LIN {X -0.023,Y -549.868,Z 969.397,A 0.000,B 0.000,C 90.000,E1 107.457} C_DIS
LIN {X -0.196,Y -549.764,Z 969.394,A 0.000,B 0.000,C 90.000,E1 106.913} C_DIS
LIN {X -0.171,Y -550.290,Z 969.388,A 0.000,B 0.000,C 90.000,E1 105.788} C_DIS
LIN {X 0.267,Y -551.658,Z 969.372,A 0.000,B 0.000,C 90.000,E1 102.939} C_DIS
LIN {X -0.148,Y -554.267,Z 969.355,A 0.000,B 0.000,C 90.000,E1 99.905} C_DIS
LIN {X -0.028,Y -555.925,Z 969.346,A 0.000,B 0.000,C 90.000,E1 98.219} C_DIS
LIN {X -0.088,Y -557.183,Z 969.338,A 0.000,B 0.000,C 90.000,E1 96.834} C_DIS
LIN {X -0.131,Y -558.262,Z 969.330,A 0.000,B 0.000,C 90.000,E1 95.448} C_DIS
LIN {X 0.223,Y -559.010,Z 969.324,A 0.000,B 0.000,C 90.000,E1 94.302} C_DIS
LIN {X 0.157,Y -559.871,Z 969.316,A 0.000,B 0.000,C 90.000,E1 92.922} C_DIS
LIN {X 0.071,Y -560.596,Z 969.309,A 0.000,B 0.000,C 90.000,E1 91.547} C_DIS
LIN {X -0.014,Y -561.277,Z 969.301,A 0.000,B 0.000,C 90.000,E1 90.172} C_DIS
LIN {X -0.086,Y -561.729,Z 969.293,A 0.000,B 0.000,C 90.000,E1 88.797} C_DIS
LIN {X -0.140,Y -562.027,Z 969.286,A 0.000,B 0.000,C 90.000,E1 87.421} C_DIS
LIN {X -0.191,Y -562.284,Z 969.278,A 0.000,B 0.000,C 90.000,E1 86.045} C_DIS
LIN {X -0.059,Y -562.524,Z 969.269,A 0.000,B 0.000,C 90.000,E1 84.375} C_DIS
LIN {X -0.068,Y -562.691,Z 969.261,A 0.000,B 0.000,C 90.000,E1 82.996} C_DIS
LIN {X -0.263,Y -563.143,Z 969.250,A 0.000,B 0.000,C 90.000,E1 81.084} C_DIS
LIN {X -0.020,Y -564.090,Z 969.237,A 0.000,B 0.000,C 90.000,E1 78.578} C_DIS
LIN {X 0.033,Y -565.125,Z 969.226,A 0.000,B 0.000,C 90.000,E1 76.645} C_DIS
LIN {X 0.068,Y -566.236,Z 969.217,A 0.000,B 0.000,C 90.000,E1 74.991} C_DIS
LIN {X -0.109,Y -567.560,Z 969.206,A 0.000,B 0.000,C 90.000,E1 73.087} C_DIS
LIN {X 0.129,Y -568.448,Z 969.198,A 0.000,B 0.000,C 90.000,E1 71.692} C_DIS
LIN {X 0.049,Y -569.047,Z 969.192,A 0.000,B 0.000,C 90.000,E1 70.604} C_DIS
LIN {X -0.030,Y -569.624,Z 969.186,A 0.000,B 0.000,C 90.000,E1 69.518} C_DIS
LIN {X -0.086,Y -570.280,Z 969.179,A 0.000,B 0.000,C 90.000,E1 68.156} C_DIS
LIN {X 0.054,Y -570.978,Z 969.168,A 0.000,B 0.000,C 90.000,E1 66.230} C_DIS
LIN {X 0.085,Y -571.434,Z 969.159,A 0.000,B 0.000,C 90.000,E1 64.588} C_DIS
LIN {X -0.228,Y -571.757,Z 969.151,A 0.000,B 0.000,C 90.000,E1 63.256} C_DIS
LIN {X -0.281,Y -571.994,Z 969.144,A 0.000,B 0.000,C 90.000,E1 61.897} C_DIS
LIN {X -0.054,Y -572.126,Z 969.136,A 0.000,B 0.000,C 90.000,E1 60.511} C_DIS
LIN {X -0.165,Y -572.288,Z 969.126,A 0.000,B 0.000,C 90.000,E1 58.614} C_DIS
LIN {X 0.003,Y -572.425,Z 969.117,A 0.000,B 0.000,C 90.000,E1 56.962} C_DIS
LIN {X 0.046,Y -572.265,Z 969.109,A 0.000,B 0.000,C 90.000,E1 55.595} C_DIS
LIN {X 0.130,Y -572.183,Z 969.104,A 0.000,B 0.000,C 90.000,E1 54.769} C_DIS
LIN {X -0.119,Y -571.801,Z 969.098,A 0.000,B 0.000,C 90.000,E1 53.703} C_DIS
LIN {X 0.293,Y -571.456,Z 969.094,A 0.000,B 0.000,C 90.000,E1 52.844} C_DIS
LIN {X -0.104,Y -570.939,Z 969.089,A 0.000,B 0.000,C 90.000,E1 52.065} C_DIS
LIN {X 0.104,Y -569.932,Z 969.082,A 0.000,B 0.000,C 90.000,E1 50.678} C_DIS
LIN {X 0.097,Y -568.784,Z 969.076,A 0.000,B 0.000,C 90.000,E1 49.585} C_DIS
LIN {X 0.027,Y -567.827,Z 969.071,A 0.000,B 0.000,C 90.000,E1 48.771} C_DIS
LIN {X -0.062,Y -566.696,Z 969.066,A 0.000,B 0.000,C 90.000,E1 47.957} C_DIS
LIN {X -0.203,Y -565.370,Z 969.062,A 0.000,B 0.000,C 90.000,E1 47.148} C_DIS
LIN {X -0.033,Y -564.399,Z 969.059,A 0.000,B 0.000,C 90.000,E1 46.581} C_DIS
LIN {X -0.027,Y -561.491,Z 969.051,A 0.000,B 0.000,C 90.000,E1 45.202} C_DIS
LIN {X 0.184,Y -559.483,Z 969.047,A 0.000,B 0.000,C 90.000,E1 44.352} C_DIS
LIN {X -0.025,Y -557.111,Z 969.042,A 0.000,B 0.000,C 90.000,E1 43.542} C_DIS
LIN {X 0.146,Y -554.460,Z 969.037,A 0.000,B 0.000,C 90.000,E1 42.690} C_DIS
LIN {X 0.288,Y -551.523,Z 969.033,A 0.000,B 0.000,C 90.000,E1 41.838} C_DIS
LIN {X -0.016,Y -549.373,Z 969.030,A 0.000,B 0.000,C 90.000,E1 41.310} C_DIS
LIN {X 0.027,Y -547.039,Z 969.026,A 0.000,B 0.000,C 90.000,E1 40.744} C_DIS
LIN {X -0.244,Y -541.935,Z 969.020,A 0.000,B 0.000,C 90.000,E1 39.644} C_DIS
LIN {X 0.162,Y -537.549,Z 969.015,A 0.000,B 0.000,C 90.000,E1 38.749} C_DIS
LIN {X 0.182,Y -532.876,Z 969.011,A 0.000,B 0.000,C 90.000,E1 37.890} C_DIS
LIN {X 0.154,Y -527.896,Z 969.006,A 0.000,B 0.000,C 90.000,E1 37.030} C_DIS
LIN {X 0.207,Y -521.789,Z 969.000,A 0.000,B 0.000,C 90.000,E1 36.011} C_DIS
LIN {X 0.112,Y -518.131,Z 968.997,A 0.000,B 0.000,C 90.000,E1 35.438} C_DIS
LIN {X 0.047,Y -512.314,Z 968.992,A 0.000,B 0.000,C 90.000,E1 34.565} C_DIS
LIN {X -0.019,Y -507.007,Z 968.988,A 0.000,B 0.000,C 90.000,E1 33.833} C_DIS
LIN {X -0.002,Y -501.298,Z 968.984,A 0.000,B 0.000,C 90.000,E1 33.086} C_DIS
LIN {X 0.100,Y -497.644,Z 968.981,A 0.000,B 0.000,C 90.000,E1 32.625} C_DIS
LIN {X -0.236,Y -493.784,Z 968.979,A 0.000,B 0.000,C 90.000,E1 32.212} C_DIS
LIN {X 0.054,Y -485.973,Z 968.974,A 0.000,B 0.000,C 90.000,E1 31.337} C_DIS
LIN {X -0.221,Y -480.273,Z 968.971,A 0.000,B 0.000,C 90.000,E1 30.797} C_DIS
LIN {X 0.069,Y -471.888,Z 968.966,A 0.000,B 0.000,C 90.000,E1 29.951} C_DIS
LIN {X -0.039,Y -461.755,Z 968.961,A 0.000,B 0.000,C 90.000,E1 29.027} C_DIS
LIN {X 0.120,Y -451.489,Z 968.956,A 0.000,B 0.000,C 90.000,E1 28.103} C_DIS
LIN {X 0.116,Y -436.406,Z 968.949,A 0.000,B 0.000,C 90.000,E1 26.821} C_DIS
LIN {X 0.074,Y -416.976,Z 968.939,A 0.000,B 0.000,C 90.000,E1 25.079} C_DIS
LIN {X 0.121,Y -403.934,Z 968.932,A 0.000,B 0.000,C 90.000,E1 23.770} C_DIS
LIN {X -0.172,Y -398.411,Z 968.929,A 0.000,B 0.000,C 90.000,E1 23.206} C_DIS
LIN {X 0.109,Y -395.804,Z 968.927,A 0.000,B 0.000,C 90.000,E1 22.845} C_DIS
LIN {X 0.092,Y -393.284,Z 968.925,A 0.000,B 0.000,C 90.000,E1 22.461} C_DIS
LIN {X 0.119,Y -392.305,Z 968.924,A 0.000,B 0.000,C 90.000,E1 22.280} C_DIS
LIN {X -0.046,Y -391.014,Z 968.922,A 0.000,B 0.000,C 90.000,E1 21.950} C_DIS
LIN {X -0.023,Y -390.506,Z 968.921,A 0.000,B 0.000,C 90.000,E1 21.770} C_DIS
LIN {X 0.080,Y -389.820,Z 968.918,A 0.000,B 0.000,C 90.000,E1 21.227} C_DIS
LIN {X 0.173,Y -389.839,Z 968.913,A 0.000,B 0.000,C 90.000,E1 20.301} C_DIS
LIN {X 0.011,Y -391.179,Z 968.903,A 0.000,B 0.000,C 90.000,E1 18.544} C_DIS
LIN {X -0.191,Y -393.357,Z 968.891,A 0.000,B 0.000,C 90.000,E1 16.441} C_DIS
LIN {X -0.016,Y -396.359,Z 968.878,A 0.000,B 0.000,C 90.000,E1 13.939} C_DIS
LIN {X -0.057,Y -400.300,Z 968.862,A 0.000,B 0.000,C 90.000,E1 11.130} C_DIS
LIN {X -0.098,Y -405.563,Z 968.844,A 0.000,B 0.000,C 90.000,E1 7.992} C_DIS
LIN {X -0.088,Y -410.839,Z 968.829,A 0.000,B 0.000,C 90.000,E1 5.220} C_DIS
LIN {X -0.030,Y -415.911,Z 968.816,A 0.000,B 0.000,C 90.000,E1 2.808} C_DIS
LIN {X 0.139,Y -421.480,Z 968.802,A 0.000,B 0.000,C 90.000,E1 0.401} C_DIS
LIN {X 0.000,Y -422.745,Z 968.800,A 0.000,B 0.000,C 90.000,E1 360.000} C_DIS
LIN {X 0.029,Y -424.625,Z 968.798,A 0.000,B 0.000,C 90.000,E1 359.542} C_DIS
LIN {X 0.053,Y -425.384,Z 968.797,A 0.000,B 0.000,C 90.000,E1 359.370} C_DIS
LIN {X -0.103,Y -429.458,Z 968.793,A 0.000,B 0.000,C 90.000,E1 358.797} C_DIS
LIN {X 0.126,Y -430.225,Z 968.793,A 0.000,B 0.000,C 90.000,E1 358.682} C_DIS
LIN {X 0.059,Y -434.488,Z 968.791,A 0.000,B 0.000,C 90.000,E1 358.339} C_DIS
LIN {X -0.032,Y -440.318,Z 968.789,A 0.000,B 0.000,C 90.000,E1 357.993} C_DIS
LIN {X 0.099,Y -448.688,Z 968.786,A 0.000,B 0.000,C 90.000,E1 357.535} C_DIS
LIN {X 0.144,Y -465.517,Z 968.781,A 0.000,B 0.000,C 90.000,E1 356.617} C_DIS
LIN {X -0.075,Y -475.617,Z 968.778,A 0.000,B 0.000,C 90.000,E1 356.102} C_DIS
LIN {X 0.065,Y -485.654,Z 968.775,A 0.000,B 0.000,C 90.000,E1 355.527} C_DIS
LIN {X 0.020,Y -503.780,Z 968.769,A 0.000,B 0.000,C 90.000,E1 354.489} C_DIS
LIN {X 0.137,Y -510.089,Z 968.767,A 0.000,B 0.000,C 90.000,E1 354.090} C_DIS
LIN {X -0.223,Y -519.507,Z 968.764,A 0.000,B 0.000,C 90.000,E1 353.514} C_DIS
LIN {X 0.172,Y -525.754,Z 968.762,A 0.000,B 0.000,C 90.000,E1 353.053} C_DIS
LIN {X -0.135,Y -533.195,Z 968.758,A 0.000,B 0.000,C 90.000,E1 352.527} C_DIS
LIN {X -0.243,Y -540.333,Z 968.755,A 0.000,B 0.000,C 90.000,E1 351.951} C_DIS
LIN {X -0.086,Y -547.213,Z 968.752,A 0.000,B 0.000,C 90.000,E1 351.310} C_DIS
LIN {X -0.080,Y -556.131,Z 968.747,A 0.000,B 0.000,C 90.000,E1 350.387} C_DIS
LIN {X 0.141,Y -558.635,Z 968.745,A 0.000,B 0.000,C 90.000,E1 350.095} C_DIS
LIN {X 0.222,Y -564.089,Z 968.741,A 0.000,B 0.000,C 90.000,E1 349.398} C_DIS
LIN {X -0.004,Y -568.264,Z 968.738,A 0.000,B 0.000,C 90.000,E1 348.870} C_DIS
LIN {X 0.117,Y -573.079,Z 968.734,A 0.000,B 0.000,C 90.000,E1 348.173} C_DIS
LIN {X -0.164,Y -577.486,Z 968.731,A 0.000,B 0.000,C 90.000,E1 347.521} C_DIS
LIN {X 0.031,Y -581.576,Z 968.727,A 0.000,B 0.000,C 90.000,E1 346.825} C_DIS
LIN {X 0.301,Y -586.151,Z 968.722,A 0.000,B 0.000,C 90.000,E1 345.992} C_DIS
LIN {X 0.165,Y -591.857,Z 968.716,A 0.000,B 0.000,C 90.000,E1 344.936} C_DIS
LIN {X -0.090,Y -596.515,Z 968.711,A 0.000,B 0.000,C 90.000,E1 344.031} C_DIS
LIN {X 0.122,Y -600.980,Z 968.706,A 0.000,B 0.000,C 90.000,E1 343.087} C_DIS
LIN {X -0.019,Y -605.148,Z 968.701,A 0.000,B 0.000,C 90.000,E1 342.181} C_DIS
LIN {X -0.150,Y -609.583,Z 968.695,A 0.000,B 0.000,C 90.000,E1 341.148} C_DIS
LIN {X 0.101,Y -614.858,Z 968.688,A 0.000,B 0.000,C 90.000,E1 339.826} C_DIS
LIN {X 0.316,Y -618.741,Z 968.682,A 0.000,B 0.000,C 90.000,E1 338.773} C_DIS
LIN {X -0.226,Y -623.156,Z 968.675,A 0.000,B 0.000,C 90.000,E1 337.539} C_DIS
LIN {X 0.109,Y -626.452,Z 968.669,A 0.000,B 0.000,C 90.000,E1 336.485} C_DIS
LIN {X -0.089,Y -629.658,Z 968.664,A 0.000,B 0.000,C 90.000,E1 335.485} C_DIS
LIN {X 0.055,Y -633.253,Z 968.657,A 0.000,B 0.000,C 90.000,E1 334.204} C_DIS
LIN {X -0.108,Y -635.188,Z 968.653,A 0.000,B 0.000,C 90.000,E1 333.461} C_DIS
LIN {X 0.124,Y -638.244,Z 968.646,A 0.000,B 0.000,C 90.000,E1 332.180} C_DIS
LIN {X 0.204,Y -641.584,Z 968.637,A 0.000,B 0.000,C 90.000,E1 330.667} C_DIS
LIN {X 0.222,Y -643.625,Z 968.632,A 0.000,B 0.000,C 90.000,E1 329.665} C_DIS
LIN {X 0.270,Y -645.444,Z 968.626,A 0.000,B 0.000,C 90.000,E1 328.663} C_DIS
LIN {X -0.207,Y -647.060,Z 968.621,A 0.000,B 0.000,C 90.000,E1 327.709} C_DIS
LIN {X -0.190,Y -648.192,Z 968.616,A 0.000,B 0.000,C 90.000,E1 326.962} C_DIS
LIN {X -0.096,Y -649.465,Z 968.611,A 0.000,B 0.000,C 90.000,E1 325.960} C_DIS
LIN {X 0.274,Y -650.838,Z 968.604,A 0.000,B 0.000,C 90.000,E1 324.689} C_DIS
LIN {X 0.228,Y -651.725,Z 968.599,A 0.000,B 0.000,C 90.000,E1 323.703} C_DIS
LIN {X 0.117,Y -652.636,Z 968.592,A 0.000,B 0.000,C 90.000,E1 322.477} C_DIS
LIN {X 0.020,Y -653.424,Z 968.585,A 0.000,B 0.000,C 90.000,E1 321.251} C_DIS
LIN {X 0.341,Y -654.031,Z 968.578,A 0.000,B 0.000,C 90.000,E1 319.989} C_DIS
LIN {X 0.131,Y -654.735,Z 968.570,A 0.000,B 0.000,C 90.000,E1 318.528} C_DIS
LIN {X 0.278,Y -656.513,Z 968.556,A 0.000,B 0.000,C 90.000,E1 316.053} C_DIS
LIN {X 0.182,Y -657.161,Z 968.552,A 0.000,B 0.000,C 90.000,E1 315.324} C_DIS
LIN {X -0.074,Y -658.922,Z 968.540,A 0.000,B 0.000,C 90.000,E1 313.137} C_DIS
LIN {X -0.192,Y -660.209,Z 968.531,A 0.000,B 0.000,C 90.000,E1 311.676} C_DIS
LIN {X 0.217,Y -661.294,Z 968.523,A 0.000,B 0.000,C 90.000,E1 310.172} C_DIS
LIN {X -0.254,Y -662.083,Z 968.517,A 0.000,B 0.000,C 90.000,E1 308.991} C_DIS
LIN {X 0.214,Y -662.804,Z 968.510,A 0.000,B 0.000,C 90.000,E1 307.729} C_DIS
LIN {X -0.172,Y -663.190,Z 968.506,A 0.000,B 0.000,C 90.000,E1 307.030} C_DIS
LIN {X 0.395,Y -663.564,Z 968.498,A 0.000,B 0.000,C 90.000,E1 305.518} C_DIS
LIN {X -0.171,Y -664.153,Z 968.485,A 0.000,B 0.000,C 90.000,E1 303.372} C_DIS
LIN {X -0.137,Y -666.262,Z 968.465,A 0.000,B 0.000,C 90.000,E1 299.716} C_DIS
LIN {X -0.283,Y -671.532,Z 968.444,A 0.000,B 0.000,C 90.000,E1 295.848} C_DIS
LIN {X -0.069,Y -675.006,Z 968.433,A 0.000,B 0.000,C 90.000,E1 293.898} C_DIS
LIN {X -0.239,Y -676.483,Z 968.427,A 0.000,B 0.000,C 90.000,E1 292.950} C_DIS
LIN {X -0.138,Y -676.843,Z 968.425,A 0.000,B 0.000,C 90.000,E1 292.461} C_DIS
LIN {X 0.042,Y -676.976,Z 968.423,A 0.000,B 0.000,C 90.000,E1 292.206} C_DIS
LIN {X 0.149,Y -676.527,Z 968.421,A 0.000,B 0.000,C 90.000,E1 291.716} C_DIS
LIN {X 0.078,Y -676.181,Z 968.419,A 0.000,B 0.000,C 90.000,E1 291.482} C_DIS
LIN {X 0.255,Y -675.341,Z 968.418,A 0.000,B 0.000,C 90.000,E1 291.227} C_DIS
LIN {X -0.358,Y -673.515,Z 968.416,A 0.000,B 0.000,C 90.000,E1 290.918} C_DIS
LIN {X -0.273,Y -672.787,Z 968.415,A 0.000,B 0.000,C 90.000,E1 290.791} C_DIS
LIN {X -0.192,Y -671.707,Z 968.415,A 0.000,B 0.000,C 90.000,E1 290.663} C_DIS
LIN {X -0.200,Y -665.376,Z 968.412,A 0.000,B 0.000,C 90.000,E1 290.174} C_DIS
LIN {X 0.124,Y -655.560,Z 968.409,A 0.000,B 0.000,C 90.000,E1 289.523} C_DIS
LIN {X 0.073,Y -655.528,Z 968.409,A 0.000,B 0.000,C 90.000,E1 289.523} C_DIS
LIN {X 0.233,Y -654.459,Z 968.408,A 0.000,B 0.000,C 90.000,E1 289.322} C_DIS
LIN {X 0.188,Y -654.455,Z 968.407,A 0.000,B 0.000,C 90.000,E1 289.322} C_DIS
LIN {X -0.378,Y -654.595,Z 968.407,A 0.000,B 0.000,C 90.000,E1 289.214} C_DIS
LIN {X -0.334,Y -654.907,Z 968.406,A 0.000,B 0.000,C 90.000,E1 289.087} C_DIS
LIN {X 0.205,Y -656.377,Z 968.404,A 0.000,B 0.000,C 90.000,E1 288.671} C_DIS
LIN {X 0.223,Y -659.981,Z 968.400,A 0.000,B 0.000,C 90.000,E1 288.055} C_DIS
LIN {X 0.113,Y -664.359,Z 968.396,A 0.000,B 0.000,C 90.000,E1 287.330} C_DIS
LIN {X -0.014,Y -667.594,Z 968.393,A 0.000,B 0.000,C 90.000,E1 286.732} C_DIS
LIN {X -0.249,Y -670.811,Z 968.389,A 0.000,B 0.000,C 90.000,E1 286.024} C_DIS
LIN {X 0.379,Y -673.195,Z 968.385,A 0.000,B 0.000,C 90.000,E1 285.245} C_DIS
LIN {X 0.259,Y -674.519,Z 968.382,A 0.000,B 0.000,C 90.000,E1 284.773} C_DIS
LIN {X 0.097,Y -676.009,Z 968.378,A 0.000,B 0.000,C 90.000,E1 284.064} C_DIS
LIN {X -0.051,Y -677.082,Z 968.374,A 0.000,B 0.000,C 90.000,E1 283.355} C_DIS
LIN {X -0.192,Y -677.905,Z 968.370,A 0.000,B 0.000,C 90.000,E1 282.647} C_DIS
LIN {X 0.194,Y -678.389,Z 968.366,A 0.000,B 0.000,C 90.000,E1 281.895} C_DIS
LIN {X 0.107,Y -678.463,Z 968.364,A 0.000,B 0.000,C 90.000,E1 281.422} C_DIS
LIN {X -0.030,Y -678.147,Z 968.360,A 0.000,B 0.000,C 90.000,E1 280.715} C_DIS
LIN {X -0.250,Y -677.631,Z 968.357,A 0.000,B 0.000,C 90.000,E1 280.254} C_DIS
LIN {X 0.148,Y -676.315,Z 968.353,A 0.000,B 0.000,C 90.000,E1 279.500} C_DIS
LIN {X 0.034,Y -675.184,Z 968.350,A 0.000,B 0.000,C 90.000,E1 279.029} C_DIS
LIN {X -0.196,Y -673.706,Z 968.348,A 0.000,B 0.000,C 90.000,E1 278.568} C_DIS
LIN {X 0.158,Y -670.834,Z 968.344,A 0.000,B 0.000,C 90.000,E1 277.814} C_DIS
LIN {X -0.010,Y -669.837,Z 968.342,A 0.000,B 0.000,C 90.000,E1 277.587} C_DIS
LIN {X -0.271,Y -666.765,Z 968.339,A 0.000,B 0.000,C 90.000,E1 277.004} C_DIS
LIN {X 0.017,Y -663.153,Z 968.335,A 0.000,B 0.000,C 90.000,E1 276.372} C_DIS
LIN {X -0.285,Y -659.871,Z 968.333,A 0.000,B 0.000,C 90.000,E1 275.910} C_DIS
LIN {X -0.055,Y -655.056,Z 968.329,A 0.000,B 0.000,C 90.000,E1 275.277} C_DIS
LIN {X 0.135,Y -649.688,Z 968.326,A 0.000,B 0.000,C 90.000,E1 274.645} C_DIS
LIN {X -0.192,Y -646.299,Z 968.324,A 0.000,B 0.000,C 90.000,E1 274.302} C_DIS
LIN {X 0.019,Y -640.144,Z 968.320,A 0.000,B 0.000,C 90.000,E1 273.669} C_DIS
LIN {X -0.189,Y -634.950,Z 968.318,A 0.000,B 0.000,C 90.000,E1 273.212} C_DIS
LIN {X -0.154,Y -627.970,Z 968.315,A 0.000,B 0.000,C 90.000,E1 272.636} C_DIS
LIN {X 0.018,Y -623.712,Z 968.313,A 0.000,B 0.000,C 90.000,E1 272.293} C_DIS
LIN {X -0.197,Y -617.870,Z 968.310,A 0.000,B 0.000,C 90.000,E1 271.892} C_DIS
LIN {X 0.051,Y -609.892,Z 968.308,A 0.000,B 0.000,C 90.000,E1 271.375} C_DIS
LIN {X -0.138,Y -603.402,Z 968.306,A 0.000,B 0.000,C 90.000,E1 271.031} C_DIS
LIN {X 0.234,Y -598.344,Z 968.304,A 0.000,B 0.000,C 90.000,E1 270.745} C_DIS
LIN {X 0.062,Y -591.196,Z 968.303,A 0.000,B 0.000,C 90.000,E1 270.458} C_DIS
LIN {X 0.209,Y -583.942,Z 968.301,A 0.000,B 0.000,C 90.000,E1 270.172} C_DIS
LIN {X 0.135,Y -578.187,Z 968.300,A 0.000,B 0.000,C 90.000,E1 270.000} C_DIS
LIN {X -0.099,Y -570.546,Z 968.299,A 0.000,B 0.000,C 90.000,E1 269.828} C_DIS
LIN {X -0.161,Y -564.727,Z 968.298,A 0.000,B 0.000,C 90.000,E1 269.714} C_DIS
LIN {X 0.108,Y -557.088,Z 968.298,A 0.000,B 0.000,C 90.000,E1 269.599} C_DIS
LIN {X 0.078,Y -553.455,Z 968.298,A 0.000,B 0.000,C 90.000,E1 269.599} C_DIS
LIN {X 0.049,Y -546.789,Z 968.298,A 0.000,B 0.000,C 90.000,E1 269.599} C_DIS
LIN {X -0.161,Y -543.039,Z 968.297,A 0.000,B 0.000,C 90.000,E1 269.427} C_DIS
LIN {X -0.210,Y -542.978,Z 968.297,A 0.000,B 0.000,C 90.000,E1 269.427} C_DIS
LIN {X -0.108,Y -542.551,Z 968.295,A 0.000,B 0.000,C 90.000,E1 269.026} C_DIS
LIN {X 0.062,Y -541.451,Z 968.287,A 0.000,B 0.000,C 90.000,E1 267.593} C_DIS
LIN {X 0.258,Y -540.117,Z 968.276,A 0.000,B 0.000,C 90.000,E1 265.584} C_DIS
LIN {X -0.142,Y -539.070,Z 968.268,A 0.000,B 0.000,C 90.000,E1 264.204} C_DIS
LIN {X -0.028,Y -538.231,Z 968.261,A 0.000,B 0.000,C 90.000,E1 263.053} C_DIS
LIN {X 0.199,Y -536.932,Z 968.254,A 0.000,B 0.000,C 90.000,E1 261.602} C_DIS
LIN {X -0.154,Y -535.172,Z 968.244,A 0.000,B 0.000,C 90.000,E1 259.926} C_DIS
LIN {X 0.110,Y -533.460,Z 968.236,A 0.000,B 0.000,C 90.000,E1 258.465} C_DIS
LIN {X -0.179,Y -531.773,Z 968.228,A 0.000,B 0.000,C 90.000,E1 257.061} C_DIS
LIN {X -0.154,Y -529.038,Z 968.215,A 0.000,B 0.000,C 90.000,E1 254.755} C_DIS
LIN {X 0.228,Y -527.861,Z 968.209,A 0.000,B 0.000,C 90.000,E1 253.559} C_DIS
LIN {X 0.097,Y -526.279,Z 968.201,A 0.000,B 0.000,C 90.000,E1 252.127} C_DIS
LIN {X -0.074,Y -523.664,Z 968.190,A 0.000,B 0.000,C 90.000,E1 250.115} C_DIS
LIN {X -0.101,Y -522.138,Z 968.183,A 0.000,B 0.000,C 90.000,E1 248.954} C_DIS
LIN {X -0.005,Y -520.325,Z 968.175,A 0.000,B 0.000,C 90.000,E1 247.486} C_DIS
LIN {X 0.104,Y -518.614,Z 968.168,A 0.000,B 0.000,C 90.000,E1 246.305} C_DIS
LIN {X 0.061,Y -516.427,Z 968.160,A 0.000,B 0.000,C 90.000,E1 244.845} C_DIS
LIN {X 0.098,Y -513.682,Z 968.151,A 0.000,B 0.000,C 90.000,E1 243.076} C_DIS
LIN {X -0.258,Y -511.317,Z 968.142,A 0.000,B 0.000,C 90.000,E1 241.641} C_DIS
LIN {X 0.042,Y -508.807,Z 968.134,A 0.000,B 0.000,C 90.000,E1 240.127} C_DIS
LIN {X -0.034,Y -506.572,Z 968.128,A 0.000,B 0.000,C 90.000,E1 238.948} C_DIS
LIN {X -0.003,Y -503.645,Z 968.119,A 0.000,B 0.000,C 90.000,E1 237.454} C_DIS
LIN {X -0.324,Y -501.011,Z 968.113,A 0.000,B 0.000,C 90.000,E1 236.294} C_DIS
LIN {X -0.250,Y -496.854,Z 968.103,A 0.000,B 0.000,C 90.000,E1 234.482} C_DIS
LIN {X 0.159,Y -493.558,Z 968.094,A 0.000,B 0.000,C 90.000,E1 232.924} C_DIS
LIN {X 0.254,Y -489.314,Z 968.084,A 0.000,B 0.000,C 90.000,E1 231.090} C_DIS
LIN {X 0.020,Y -484.291,Z 968.072,A 0.000,B 0.000,C 90.000,E1 228.976} C_DIS
LIN {X -0.079,Y -481.495,Z 968.065,A 0.000,B 0.000,C 90.000,E1 227.757} C_DIS
LIN {X 0.239,Y -476.090,Z 968.052,A 0.000,B 0.000,C 90.000,E1 225.243} C_DIS
LIN {X 0.089,Y -472.606,Z 968.043,A 0.000,B 0.000,C 90.000,E1 223.704} C_DIS
LIN {X 0.127,Y -469.852,Z 968.036,A 0.000,B 0.000,C 90.000,E1 222.447} C_DIS
LIN {X -0.122,Y -466.373,Z 968.027,A 0.000,B 0.000,C 90.000,E1 220.906} C_DIS
LIN {X -0.088,Y -462.897,Z 968.018,A 0.000,B 0.000,C 90.000,E1 219.322} C_DIS
LIN {X 0.068,Y -457.949,Z 968.006,A 0.000,B 0.000,C 90.000,E1 217.076} C_DIS
LIN {X 0.105,Y -454.372,Z 967.997,A 0.000,B 0.000,C 90.000,E1 215.471} C_DIS
LIN {X -0.123,Y -449.437,Z 967.985,A 0.000,B 0.000,C 90.000,E1 213.245} C_DIS
LIN {X 0.254,Y -444.521,Z 967.972,A 0.000,B 0.000,C 90.000,E1 210.924} C_DIS
LIN {X -0.120,Y -441.694,Z 967.965,A 0.000,B 0.000,C 90.000,E1 209.667} C_DIS
LIN {X -0.114,Y -438.081,Z 967.956,A 0.000,B 0.000,C 90.000,E1 208.025} C_DIS
LIN {X 0.004,Y -434.516,Z 967.946,A 0.000,B 0.000,C 90.000,E1 206.360} C_DIS
LIN {X 0.051,Y -431.526,Z 967.939,A 0.000,B 0.000,C 90.000,E1 205.027} C_DIS
LIN {X 0.046,Y -428.425,Z 967.932,A 0.000,B 0.000,C 90.000,E1 203.695} C_DIS
LIN {X -0.198,Y -423.829,Z 967.921,A 0.000,B 0.000,C 90.000,E1 201.716} C_DIS
LIN {X 0.240,Y -419.583,Z 967.909,A 0.000,B 0.000,C 90.000,E1 199.631} C_DIS
LIN {X 0.198,Y -414.058,Z 967.894,A 0.000,B 0.000,C 90.000,E1 196.913} C_DIS
LIN {X -0.112,Y -410.160,Z 967.883,A 0.000,B 0.000,C 90.000,E1 194.898} C_DIS
LIN {X -0.123,Y -406.789,Z 967.873,A 0.000,B 0.000,C 90.000,E1 193.175} C_DIS
LIN {X 0.006,Y -403.417,Z 967.864,A 0.000,B 0.000,C 90.000,E1 191.422} C_DIS
LIN {X 0.067,Y -400.132,Z 967.854,A 0.000,B 0.000,C 90.000,E1 189.670} C_DIS
LIN {X -0.071,Y -396.766,Z 967.844,A 0.000,B 0.000,C 90.000,E1 187.936} C_DIS
LIN {X -0.099,Y -391.336,Z 967.826,A 0.000,B 0.000,C 90.000,E1 184.759} C_DIS
LIN {X 0.147,Y -390.427,Z 967.822,A 0.000,B 0.000,C 90.000,E1 184.012} C_DIS
LIN {X -0.095,Y -389.546,Z 967.817,A 0.000,B 0.000,C 90.000,E1 182.980} C_DIS
LIN {X 0.115,Y -389.401,Z 967.813,A 0.000,B 0.000,C 90.000,E1 182.236} C_DIS
LIN {X 0.027,Y -389.580,Z 967.811,A 0.000,B 0.000,C 90.000,E1 181.892} C_DIS
LIN {X -0.050,Y -389.919,Z 967.809,A 0.000,B 0.000,C 90.000,E1 181.547} C_DIS
LIN {X -0.183,Y -390.765,Z 967.806,A 0.000,B 0.000,C 90.000,E1 181.031} C_DIS
LIN {X 0.082,Y -392.364,Z 967.803,A 0.000,B 0.000,C 90.000,E1 180.458} C_DIS
LIN {X 0.013,Y -394.530,Z 967.800,A 0.000,B 0.000,C 90.000,E1 179.943} C_DIS
LIN {X -0.050,Y -399.098,Z 967.796,A 0.000,B 0.000,C 90.000,E1 179.198} C_DIS
LIN {X -0.099,Y -405.521,Z 967.791,A 0.000,B 0.000,C 90.000,E1 178.453} C_DIS
LIN {X 0.081,Y -411.802,Z 967.788,A 0.000,B 0.000,C 90.000,E1 177.822} C_DIS
LIN {X -0.203,Y -419.334,Z 967.784,A 0.000,B 0.000,C 90.000,E1 177.192} C_DIS
LIN {X 0.072,Y -431.410,Z 967.778,A 0.000,B 0.000,C 90.000,E1 176.045} C_DIS
LIN {X -0.133,Y -443.385,Z 967.772,A 0.000,B 0.000,C 90.000,E1 174.951} C_DIS
LIN {X 0.180,Y -451.803,Z 967.767,A 0.000,B 0.000,C 90.000,E1 174.090} C_DIS
LIN {X -0.027,Y -458.927,Z 967.763,A 0.000,B 0.000,C 90.000,E1 173.394} C_DIS
LIN {X 0.065,Y -465.739,Z 967.759,A 0.000,B 0.000,C 90.000,E1 172.648} C_DIS
LIN {X 0.018,Y -472.498,Z 967.755,A 0.000,B 0.000,C 90.000,E1 171.894} C_DIS
LIN {X -0.232,Y -480.101,Z 967.750,A 0.000,B 0.000,C 90.000,E1 171.027} C_DIS
LIN {X 0.200,Y -489.846,Z 967.743,A 0.000,B 0.000,C 90.000,E1 169.746} C_DIS
LIN {X 0.031,Y -497.947,Z 967.737,A 0.000,B 0.000,C 90.000,E1 168.701} C_DIS
LIN {X 0.062,Y -505.525,Z 967.731,A 0.000,B 0.000,C 90.000,E1 167.645} C_DIS
LIN {X 0.023,Y -511.685,Z 967.727,A 0.000,B 0.000,C 90.000,E1 166.756} C_DIS
LIN {X -0.013,Y -513.742,Z 967.725,A 0.000,B 0.000,C 90.000,E1 166.464} C_DIS
LIN {X -0.291,Y -522.062,Z 967.717,A 0.000,B 0.000,C 90.000,E1 165.172} C_DIS
LIN {X 0.012,Y -529.357,Z 967.711,A 0.000,B 0.000,C 90.000,E1 163.976} C_DIS
LIN {X 0.121,Y -537.301,Z 967.704,A 0.000,B 0.000,C 90.000,E1 162.670} C_DIS
LIN {X -0.210,Y -548.220,Z 967.694,A 0.000,B 0.000,C 90.000,E1 160.859} C_DIS
LIN {X 0.146,Y -554.756,Z 967.687,A 0.000,B 0.000,C 90.000,E1 159.699} C_DIS
LIN {X -0.024,Y -561.770,Z 967.680,A 0.000,B 0.000,C 90.000,E1 158.465} C_DIS
LIN {X 0.105,Y -566.926,Z 967.675,A 0.000,B 0.000,C 90.000,E1 157.486} C_DIS
LIN {X 0.078,Y -571.194,Z 967.670,A 0.000,B 0.000,C 90.000,E1 156.666} C_DIS
LIN {X 0.078,Y -577.855,Z 967.663,A 0.000,B 0.000,C 90.000,E1 155.305} C_DIS
LIN {X -0.359,Y -581.485,Z 967.658,A 0.000,B 0.000,C 90.000,E1 154.537} C_DIS
LIN {X -0.105,Y -585.984,Z 967.652,A 0.000,B 0.000,C 90.000,E1 153.435} C_DIS
LIN {X -0.050,Y -590.172,Z 967.646,A 0.000,B 0.000,C 90.000,E1 152.359} C_DIS
LIN {X -0.190,Y -593.854,Z 967.641,A 0.000,B 0.000,C 90.000,E1 151.307} C_DIS
LIN {X 0.367,Y -599.028,Z 967.632,A 0.000,B 0.000,C 90.000,E1 149.665} C_DIS
LIN {X -0.167,Y -602.444,Z 967.626,A 0.000,B 0.000,C 90.000,E1 148.663} C_DIS
LIN {X 0.103,Y -606.702,Z 967.619,A 0.000,B 0.000,C 90.000,E1 147.327} C_DIS
LIN {X -0.011,Y -609.910,Z 967.613,A 0.000,B 0.000,C 90.000,E1 146.294} C_DIS
LIN {X -0.082,Y -613.296,Z 967.607,A 0.000,B 0.000,C 90.000,E1 145.261} C_DIS
LIN {X -0.003,Y -618.249,Z 967.598,A 0.000,B 0.000,C 90.000,E1 143.703} C_DIS
LIN {X 0.012,Y -623.840,Z 967.588,A 0.000,B 0.000,C 90.000,E1 141.904} C_DIS
LIN {X -0.151,Y -627.845,Z 967.581,A 0.000,B 0.000,C 90.000,E1 140.642} C_DIS
LIN {X -0.246,Y -631.776,Z 967.574,A 0.000,B 0.000,C 90.000,E1 139.380} C_DIS
LIN {X 0.304,Y -638.188,Z 967.563,A 0.000,B 0.000,C 90.000,E1 137.310} C_DIS
LIN {X 0.326,Y -642.327,Z 967.556,A 0.000,B 0.000,C 90.000,E1 136.053} C_DIS
LIN {X -0.113,Y -647.370,Z 967.548,A 0.000,B 0.000,C 90.000,E1 134.595} C_DIS
LIN {X -0.036,Y -653.433,Z 967.538,A 0.000,B 0.000,C 90.000,E1 132.852} C_DIS
LIN {X 0.172,Y -661.554,Z 967.526,A 0.000,B 0.000,C 90.000,E1 130.620} C_DIS
LIN {X 0.136,Y -666.155,Z 967.519,A 0.000,B 0.000,C 90.000,E1 129.402} C_DIS
LIN {X -0.246,Y -669.688,Z 967.514,A 0.000,B 0.000,C 90.000,E1 128.463} C_DIS
LIN {X -0.057,Y -674.761,Z 967.506,A 0.000,B 0.000,C 90.000,E1 126.996} C_DIS
LIN {X 0.213,Y -677.875,Z 967.500,A 0.000,B 0.000,C 90.000,E1 126.011} C_DIS
LIN {X 0.139,Y -681.585,Z 967.494,A 0.000,B 0.000,C 90.000,E1 124.818} C_DIS
LIN {X 0.117,Y -684.390,Z 967.488,A 0.000,B 0.000,C 90.000,E1 123.865} C_DIS
LIN {X -0.437,Y -687.004,Z 967.483,A 0.000,B 0.000,C 90.000,E1 122.959} C_DIS
LIN {X -0.387,Y -689.468,Z 967.478,A 0.000,B 0.000,C 90.000,E1 122.005} C_DIS
LIN {X 0.280,Y -691.807,Z 967.472,A 0.000,B 0.000,C 90.000,E1 121.003} C_DIS
LIN {X 0.035,Y -693.923,Z 967.467,A 0.000,B 0.000,C 90.000,E1 120.079} C_DIS
LIN {X -0.434,Y -695.321,Z 967.463,A 0.000,B 0.000,C 90.000,E1 119.411} C_DIS
LIN {X -0.029,Y -696.629,Z 967.458,A 0.000,B 0.000,C 90.000,E1 118.437} C_DIS
LIN {X 0.039,Y -697.909,Z 967.451,A 0.000,B 0.000,C 90.000,E1 117.257} C_DIS
LIN {X 0.161,Y -698.707,Z 967.446,A 0.000,B 0.000,C 90.000,E1 116.309} C_DIS
LIN {X -0.330,Y -699.277,Z 967.441,A 0.000,B 0.000,C 90.000,E1 115.412} C_DIS
LIN {X -0.161,Y -699.520,Z 967.437,A 0.000,B 0.000,C 90.000,E1 114.695} C_DIS
LIN {X 0.081,Y -699.511,Z 967.435,A 0.000,B 0.000,C 90.000,E1 114.207} C_DIS
LIN {X -0.308,Y -699.164,Z 967.432,A 0.000,B 0.000,C 90.000,E1 113.770} C_DIS
LIN {X -0.042,Y -698.683,Z 967.431,A 0.000,B 0.000,C 90.000,E1 113.515} C_DIS
LIN {X 0.207,Y -697.286,Z 967.428,A 0.000,B 0.000,C 90.000,E1 113.025} C_DIS
LIN {X -0.306,Y -696.683,Z 967.427,A 0.000,B 0.000,C 90.000,E1 112.950} C_DIS
LIN {X -0.194,Y -693.909,Z 967.425,A 0.000,B 0.000,C 90.000,E1 112.589} C_DIS
LIN {X 0.051,Y -691.862,Z 967.424,A 0.000,B 0.000,C 90.000,E1 112.333} C_DIS
LIN {X 0.170,Y -690.258,Z 967.424,A 0.000,B 0.000,C 90.000,E1 112.206} C_DIS
LIN {X 0.045,Y -685.997,Z 967.422,A 0.000,B 0.000,C 90.000,E1 112.025} C_DIS
LIN {X -0.056,Y -682.203,Z 967.422,A 0.000,B 0.000,C 90.000,E1 111.897} C_DIS
LIN {X 0.140,Y -676.018,Z 967.421,A 0.000,B 0.000,C 90.000,E1 111.716} C_DIS
LIN {X -0.109,Y -674.262,Z 967.421,A 0.000,B 0.000,C 90.000,E1 111.716} C_DIS
LIN {X 0.226,Y -667.115,Z 967.421,A 0.000,B 0.000,C 90.000,E1 111.663} C_DIS
LIN {X 0.167,Y -627.310,Z 967.420,A 0.000,B 0.000,C 90.000,E1 111.663} C_DIS
LIN {X 0.224,Y -622.838,Z 967.420,A 0.000,B 0.000,C 90.000,E1 111.589} C_DIS
LIN {X -0.100,Y -616.034,Z 967.419,A 0.000,B 0.000,C 90.000,E1 111.461} C_DIS
LIN {X -0.055,Y -609.075,Z 967.418,A 0.000,B 0.000,C 90.000,E1 111.227} C_DIS
LIN {X -0.202,Y -604.447,Z 967.417,A 0.000,B 0.000,C 90.000,E1 111.046} C_DIS
LIN {X 0.226,Y -599.289,Z 967.415,A 0.000,B 0.000,C 90.000,E1 110.737} C_DIS
LIN {X -0.097,Y -592.629,Z 967.413,A 0.000,B 0.000,C 90.000,E1 110.355} C_DIS
LIN {X 0.329,Y -583.313,Z 967.409,A 0.000,B 0.000,C 90.000,E1 109.631} C_DIS
LIN {X 0.207,Y -576.121,Z 967.406,A 0.000,B 0.000,C 90.000,E1 109.087} C_DIS
LIN {X -0.176,Y -574.529,Z 967.406,A 0.000,B 0.000,C 90.000,E1 109.014} C_DIS
LIN {X -0.017,Y -567.870,Z 967.403,A 0.000,B 0.000,C 90.000,E1 108.598} C_DIS
LIN {X 0.198,Y -552.790,Z 967.399,A 0.000,B 0.000,C 90.000,E1 107.819} C_DIS
LIN {X -0.111,Y -550.419,Z 967.398,A 0.000,B 0.000,C 90.000,E1 107.638} C_DIS
LIN {X -0.149,Y -550.391,Z 967.398,A 0.000,B 0.000,C 90.000,E1 107.638} C_DIS
LIN {X 0.177,Y -549.932,Z 967.397,A 0.000,B 0.000,C 90.000,E1 107.402} C_DIS
LIN {X -0.099,Y -549.969,Z 967.393,A 0.000,B 0.000,C 90.000,E1 106.732} C_DIS
LIN {X -0.072,Y -550.481,Z 967.387,A 0.000,B 0.000,C 90.000,E1 105.607} C_DIS
LIN {X 0.127,Y -551.713,Z 967.373,A 0.000,B 0.000,C 90.000,E1 103.063} C_DIS
LIN {X -0.051,Y -554.530,Z 967.354,A 0.000,B 0.000,C 90.000,E1 99.726} C_DIS
LIN {X 0.117,Y -556.419,Z 967.343,A 0.000,B 0.000,C 90.000,E1 97.757} C_DIS
LIN {X -0.062,Y -557.382,Z 967.337,A 0.000,B 0.000,C 90.000,E1 96.663} C_DIS
LIN {X -0.098,Y -558.452,Z 967.329,A 0.000,B 0.000,C 90.000,E1 95.277} C_DIS
LIN {X 0.263,Y -559.156,Z 967.323,A 0.000,B 0.000,C 90.000,E1 94.131} C_DIS
LIN {X 0.202,Y -560.000,Z 967.315,A 0.000,B 0.000,C 90.000,E1 92.751} C_DIS
LIN {X 0.213,Y -560.869,Z 967.306,A 0.000,B 0.000,C 90.000,E1 91.088} C_DIS
LIN {X 0.134,Y -561.465,Z 967.299,A 0.000,B 0.000,C 90.000,E1 89.714} C_DIS
LIN {X 0.063,Y -561.870,Z 967.291,A 0.000,B 0.000,C 90.000,E1 88.339} C_DIS
LIN {X 0.136,Y -562.204,Z 967.282,A 0.000,B 0.000,C 90.000,E1 86.674} C_DIS
LIN {X 0.087,Y -562.410,Z 967.274,A 0.000,B 0.000,C 90.000,E1 85.298} C_DIS
LIN {X 0.136,Y -562.633,Z 967.266,A 0.000,B 0.000,C 90.000,E1 83.913} C_DIS
LIN {X -0.051,Y -563.002,Z 967.254,A 0.000,B 0.000,C 90.000,E1 81.724} C_DIS
LIN {X -0.144,Y -563.570,Z 967.243,A 0.000,B 0.000,C 90.000,E1 79.803} C_DIS
LIN {X -0.218,Y -564.484,Z 967.233,A 0.000,B 0.000,C 90.000,E1 77.881} C_DIS
LIN {X 0.133,Y -565.807,Z 967.220,A 0.000,B 0.000,C 90.000,E1 75.644} C_DIS
LIN {X -0.053,Y -567.121,Z 967.210,A 0.000,B 0.000,C 90.000,E1 73.740} C_DIS
LIN {X 0.005,Y -568.048,Z 967.202,A 0.000,B 0.000,C 90.000,E1 72.362} C_DIS
LIN {X -0.126,Y -569.029,Z 967.193,A 0.000,B 0.000,C 90.000,E1 70.732} C_DIS
LIN {X 0.138,Y -569.701,Z 967.185,A 0.000,B 0.000,C 90.000,E1 69.337} C_DIS
LIN {X 0.082,Y -570.331,Z 967.178,A 0.000,B 0.000,C 90.000,E1 67.975} C_DIS
LIN {X 0.218,Y -571.002,Z 967.167,A 0.000,B 0.000,C 90.000,E1 66.049} C_DIS
LIN {X 0.245,Y -571.396,Z 967.158,A 0.000,B 0.000,C 90.000,E1 64.409} C_DIS
LIN {X -0.075,Y -571.717,Z 967.150,A 0.000,B 0.000,C 90.000,E1 63.076} C_DIS
LIN {X -0.136,Y -571.932,Z 967.143,A 0.000,B 0.000,C 90.000,E1 61.719} C_DIS
LIN {X 0.083,Y -572.044,Z 967.135,A 0.000,B 0.000,C 90.000,E1 60.333} C_DIS
LIN {X -0.184,Y -572.179,Z 967.128,A 0.000,B 0.000,C 90.000,E1 58.997} C_DIS
LIN {X 0.339,Y -572.294,Z 967.120,A 0.000,B 0.000,C 90.000,E1 57.582} C_DIS
LIN {X 0.113,Y -572.300,Z 967.116,A 0.000,B 0.000,C 90.000,E1 56.786} C_DIS
LIN {X -0.004,Y -572.115,Z 967.108,A 0.000,B 0.000,C 90.000,E1 55.435} C_DIS
LIN {X 0.082,Y -571.976,Z 967.103,A 0.000,B 0.000,C 90.000,E1 54.609} C_DIS
LIN {X 0.022,Y -571.868,Z 967.100,A 0.000,B 0.000,C 90.000,E1 54.069} C_DIS
LIN {X 0.111,Y -571.359,Z 967.094,A 0.000,B 0.000,C 90.000,E1 52.970} C_DIS
LIN {X -0.283,Y -570.858,Z 967.090,A 0.000,B 0.000,C 90.000,E1 52.190} C_DIS
LIN {X -0.069,Y -569.815,Z 967.082,A 0.000,B 0.000,C 90.000,E1 50.803} C_DIS
LIN {X -0.008,Y -568.693,Z 967.076,A 0.000,B 0.000,C 90.000,E1 49.703} C_DIS
LIN {X -0.023,Y -567.363,Z 967.070,A 0.000,B 0.000,C 90.000,E1 48.609} C_DIS
LIN {X -0.049,Y -565.736,Z 967.064,A 0.000,B 0.000,C 90.000,E1 47.514} C_DIS
LIN {X 0.314,Y -563.722,Z 967.058,A 0.000,B 0.000,C 90.000,E1 46.377} C_DIS
LIN {X -0.324,Y -562.595,Z 967.055,A 0.000,B 0.000,C 90.000,E1 45.891} C_DIS
LIN {X 0.296,Y -560.732,Z 967.050,A 0.000,B 0.000,C 90.000,E1 45.000} C_DIS
LIN {X 0.102,Y -558.590,Z 967.046,A 0.000,B 0.000,C 90.000,E1 44.190} C_DIS
LIN {X -0.115,Y -556.135,Z 967.041,A 0.000,B 0.000,C 90.000,E1 43.380} C_DIS
LIN {X 0.044,Y -553.399,Z 967.036,A 0.000,B 0.000,C 90.000,E1 42.528} C_DIS
LIN {X -0.248,Y -551.394,Z 967.033,A 0.000,B 0.000,C 90.000,E1 42.000} C_DIS
LIN {X -0.136,Y -548.146,Z 967.029,A 0.000,B 0.000,C 90.000,E1 41.148} C_DIS
LIN {X -0.264,Y -545.063,Z 967.025,A 0.000,B 0.000,C 90.000,E1 40.458} C_DIS
LIN {X -0.006,Y -541.829,Z 967.021,A 0.000,B 0.000,C 90.000,E1 39.725} C_DIS
LIN {X -0.184,Y -536.672,Z 967.015,A 0.000,B 0.000,C 90.000,E1 38.749} C_DIS
LIN {X -0.171,Y -531.920,Z 967.010,A 0.000,B 0.000,C 90.000,E1 37.890} C_DIS
LIN {X 0.113,Y -526.875,Z 967.006,A 0.000,B 0.000,C 90.000,E1 36.996} C_DIS
LIN {X -0.159,Y -520.696,Z 967.000,A 0.000,B 0.000,C 90.000,E1 36.011} C_DIS
LIN {X 0.101,Y -515.084,Z 966.995,A 0.000,B 0.000,C 90.000,E1 35.105} C_DIS
LIN {X -0.228,Y -510.035,Z 966.991,A 0.000,B 0.000,C 90.000,E1 34.405} C_DIS
LIN {X 0.103,Y -504.514,Z 966.987,A 0.000,B 0.000,C 90.000,E1 33.627} C_DIS
LIN {X 0.023,Y -499.837,Z 966.984,A 0.000,B 0.000,C 90.000,E1 33.038} C_DIS
LIN {X -0.021,Y -493.605,Z 966.979,A 0.000,B 0.000,C 90.000,E1 32.291} C_DIS
LIN {X 0.238,Y -484.140,Z 966.974,A 0.000,B 0.000,C 90.000,E1 31.258} C_DIS
LIN {X -0.096,Y -476.951,Z 966.970,A 0.000,B 0.000,C 90.000,E1 30.590} C_DIS
LIN {X 0.062,Y -468.229,Z 966.965,A 0.000,B 0.000,C 90.000,E1 29.745} C_DIS
LIN {X 0.037,Y -462.348,Z 966.962,A 0.000,B 0.000,C 90.000,E1 29.205} C_DIS
LIN {X 0.024,Y -453.290,Z 966.958,A 0.000,B 0.000,C 90.000,E1 28.409} C_DIS
LIN {X -0.123,Y -441.071,Z 966.952,A 0.000,B 0.000,C 90.000,E1 27.385} C_DIS
LIN {X 0.169,Y -416.994,Z 966.940,A 0.000,B 0.000,C 90.000,E1 25.207} C_DIS
LIN {X -0.033,Y -402.378,Z 966.932,A 0.000,B 0.000,C 90.000,E1 23.770} C_DIS
LIN {X -0.192,Y -398.273,Z 966.930,A 0.000,B 0.000,C 90.000,E1 23.334} C_DIS
LIN {X 0.081,Y -396.073,Z 966.928,A 0.000,B 0.000,C 90.000,E1 23.025} C_DIS
LIN {X -0.203,Y -392.270,Z 966.925,A 0.000,B 0.000,C 90.000,E1 22.461} C_DIS
LIN {X -0.107,Y -390.513,Z 966.922,A 0.000,B 0.000,C 90.000,E1 21.950} C_DIS
LIN {X 0.220,Y -389.751,Z 966.918,A 0.000,B 0.000,C 90.000,E1 21.280} C_DIS
LIN {X 0.150,Y -389.747,Z 966.914,A 0.000,B 0.000,C 90.000,E1 20.556} C_DIS
LIN {X 0.035,Y -390.410,Z 966.908,A 0.000,B 0.000,C 90.000,E1 19.504} C_DIS
LIN {X -0.096,Y -393.983,Z 966.889,A 0.000,B 0.000,C 90.000,E1 15.969} C_DIS
LIN {X 0.040,Y -396.607,Z 966.877,A 0.000,B 0.000,C 90.000,E1 13.828} C_DIS
LIN {X 0.078,Y -401.105,Z 966.859,A 0.000,B 0.000,C 90.000,E1 10.658} C_DIS
LIN {X 0.050,Y -405.842,Z 966.844,A 0.000,B 0.000,C 90.000,E1 7.871} C_DIS
LIN {X -0.002,Y -410.468,Z 966.830,A 0.000,B 0.000,C 90.000,E1 5.454} C_DIS
LIN {X 0.090,Y -416.215,Z 966.815,A 0.000,B 0.000,C 90.000,E1 2.694} C_DIS
LIN {X -0.186,Y -420.853,Z 966.804,A 0.000,B 0.000,C 90.000,E1 0.688} C_DIS
LIN {X 0.000,Y -422.713,Z 966.800,A 0.000,B 0.000,C 90.000,E1 360.000} C_DIS
LIN {X 0.033,Y -425.462,Z 966.796,A 0.000,B 0.000,C 90.000,E1 359.312} C_DIS
LIN {X 0.085,Y -427.570,Z 966.794,A 0.000,B 0.000,C 90.000,E1 358.969} C_DIS
LIN {X -0.085,Y -429.363,Z 966.793,A 0.000,B 0.000,C 90.000,E1 358.740} C_DIS
LIN {X 0.145,Y -430.132,Z 966.793,A 0.000,B 0.000,C 90.000,E1 358.625} C_DIS
LIN {X -0.042,Y -435.272,Z 966.790,A 0.000,B 0.000,C 90.000,E1 358.224} C_DIS
LIN {X -0.087,Y -441.202,Z 966.788,A 0.000,B 0.000,C 90.000,E1 357.879} C_DIS
LIN {X 0.035,Y -447.491,Z 966.786,A 0.000,B 0.000,C 90.000,E1 357.535} C_DIS
LIN {X 0.042,Y -464.462,Z 966.781,A 0.000,B 0.000,C 90.000,E1 356.617} C_DIS
LIN {X -0.169,Y -474.565,Z 966.778,A 0.000,B 0.000,C 90.000,E1 356.102} C_DIS
LIN {X -0.046,Y -487.628,Z 966.774,A 0.000,B 0.000,C 90.000,E1 355.355} C_DIS
LIN {X -0.166,Y -502.053,Z 966.770,A 0.000,B 0.000,C 90.000,E1 354.546} C_DIS
LIN {X -0.136,Y -506.871,Z 966.768,A 0.000,B 0.000,C 90.000,E1 354.261} C_DIS
LIN {X -0.237,Y -517.773,Z 966.764,A 0.000,B 0.000,C 90.000,E1 353.571} C_DIS
LIN {X -0.274,Y -525.578,Z 966.761,A 0.000,B 0.000,C 90.000,E1 353.053} C_DIS
LIN {X 0.003,Y -533.005,Z 966.758,A 0.000,B 0.000,C 90.000,E1 352.470} C_DIS
LIN {X -0.239,Y -541.561,Z 966.754,A 0.000,B 0.000,C 90.000,E1 351.781} C_DIS
LIN {X 0.030,Y -547.048,Z 966.751,A 0.000,B 0.000,C 90.000,E1 351.254} C_DIS
LIN {X 0.179,Y -554.852,Z 966.747,A 0.000,B 0.000,C 90.000,E1 350.443} C_DIS
LIN {X 0.165,Y -558.614,Z 966.745,A 0.000,B 0.000,C 90.000,E1 350.038} C_DIS
LIN {X 0.205,Y -564.176,Z 966.741,A 0.000,B 0.000,C 90.000,E1 349.342} C_DIS
LIN {X -0.021,Y -568.361,Z 966.738,A 0.000,B 0.000,C 90.000,E1 348.814} C_DIS
LIN {X -0.218,Y -572.256,Z 966.735,A 0.000,B 0.000,C 90.000,E1 348.285} C_DIS
LIN {X -0.183,Y -577.626,Z 966.730,A 0.000,B 0.000,C 90.000,E1 347.465} C_DIS
LIN {X -0.194,Y -583.300,Z 966.725,A 0.000,B 0.000,C 90.000,E1 346.520} C_DIS
LIN {X 0.059,Y -587.023,Z 966.721,A 0.000,B 0.000,C 90.000,E1 345.825} C_DIS
LIN {X 0.311,Y -592.041,Z 966.716,A 0.000,B 0.000,C 90.000,E1 344.866} C_DIS
LIN {X -0.097,Y -596.740,Z 966.711,A 0.000,B 0.000,C 90.000,E1 343.976} C_DIS
LIN {X 0.059,Y -601.798,Z 966.705,A 0.000,B 0.000,C 90.000,E1 342.906} C_DIS
LIN {X -0.073,Y -605.918,Z 966.700,A 0.000,B 0.000,C 90.000,E1 342.000} C_DIS
LIN {X -0.193,Y -610.349,Z 966.694,A 0.000,B 0.000,C 90.000,E1 340.967} C_DIS
LIN {X -0.251,Y -614.571,Z 966.688,A 0.000,B 0.000,C 90.000,E1 339.934} C_DIS
LIN {X -0.257,Y -618.520,Z 966.683,A 0.000,B 0.000,C 90.000,E1 338.901} C_DIS
LIN {X 0.013,Y -622.148,Z 966.677,A 0.000,B 0.000,C 90.000,E1 337.847} C_DIS
LIN {X 0.337,Y -625.517,Z 966.671,A 0.000,B 0.000,C 90.000,E1 336.794} C_DIS
LIN {X 0.150,Y -629.567,Z 966.664,A 0.000,B 0.000,C 90.000,E1 335.537} C_DIS
LIN {X -0.040,Y -631.776,Z 966.660,A 0.000,B 0.000,C 90.000,E1 334.793} C_DIS
LIN {X 0.100,Y -634.597,Z 966.654,A 0.000,B 0.000,C 90.000,E1 333.768} C_DIS
LIN {X -0.236,Y -637.683,Z 966.647,A 0.000,B 0.000,C 90.000,E1 332.538} C_DIS
LIN {X -0.017,Y -639.976,Z 966.642,A 0.000,B 0.000,C 90.000,E1 331.513} C_DIS
LIN {X 0.042,Y -642.758,Z 966.635,A 0.000,B 0.000,C 90.000,E1 330.255} C_DIS
LIN {X 0.081,Y -644.706,Z 966.629,A 0.000,B 0.000,C 90.000,E1 329.253} C_DIS
LIN {X 0.217,Y -646.860,Z 966.622,A 0.000,B 0.000,C 90.000,E1 327.995} C_DIS
LIN {X -0.243,Y -648.420,Z 966.617,A 0.000,B 0.000,C 90.000,E1 327.041} C_DIS
LIN {X 0.215,Y -649.704,Z 966.611,A 0.000,B 0.000,C 90.000,E1 326.008} C_DIS
LIN {X -0.245,Y -651.385,Z 966.603,A 0.000,B 0.000,C 90.000,E1 324.562} C_DIS
LIN {X 0.098,Y -652.249,Z 966.598,A 0.000,B 0.000,C 90.000,E1 323.543} C_DIS
LIN {X 0.069,Y -652.968,Z 966.592,A 0.000,B 0.000,C 90.000,E1 322.557} C_DIS
LIN {X -0.026,Y -653.804,Z 966.585,A 0.000,B 0.000,C 90.000,E1 321.331} C_DIS
LIN {X 0.299,Y -654.457,Z 966.578,A 0.000,B 0.000,C 90.000,E1 320.070} C_DIS
LIN {X 0.065,Y -655.391,Z 966.567,A 0.000,B 0.000,C 90.000,E1 318.119} C_DIS
LIN {X 0.252,Y -656.869,Z 966.556,A 0.000,B 0.000,C 90.000,E1 316.134} C_DIS
LIN {X 0.131,Y -657.706,Z 966.551,A 0.000,B 0.000,C 90.000,E1 315.162} C_DIS
LIN {X -0.085,Y -659.307,Z 966.540,A 0.000,B 0.000,C 90.000,E1 313.218} C_DIS
LIN {X -0.194,Y -660.623,Z 966.532,A 0.000,B 0.000,C 90.000,E1 311.757} C_DIS
LIN {X 0.200,Y -661.896,Z 966.522,A 0.000,B 0.000,C 90.000,E1 310.011} C_DIS
LIN {X -0.266,Y -662.685,Z 966.516,A 0.000,B 0.000,C 90.000,E1 308.830} C_DIS
LIN {X -0.198,Y -663.393,Z 966.509,A 0.000,B 0.000,C 90.000,E1 307.604} C_DIS
LIN {X 0.261,Y -663.681,Z 966.506,A 0.000,B 0.000,C 90.000,E1 307.076} C_DIS
LIN {X -0.053,Y -664.030,Z 966.499,A 0.000,B 0.000,C 90.000,E1 305.884} C_DIS
LIN {X 0.023,Y -664.268,Z 966.493,A 0.000,B 0.000,C 90.000,E1 304.659} C_DIS
LIN {X -0.167,Y -664.746,Z 966.484,A 0.000,B 0.000,C 90.000,E1 303.214} C_DIS
LIN {X -0.028,Y -666.727,Z 966.466,A 0.000,B 0.000,C 90.000,E1 299.795} C_DIS
LIN {X 0.093,Y -670.359,Z 966.449,A 0.000,B 0.000,C 90.000,E1 296.873} C_DIS
LIN {X 0.198,Y -674.975,Z 966.435,A 0.000,B 0.000,C 90.000,E1 294.207} C_DIS
LIN {X 0.027,Y -676.537,Z 966.429,A 0.000,B 0.000,C 90.000,E1 293.259} C_DIS
LIN {X 0.127,Y -677.201,Z 966.427,A 0.000,B 0.000,C 90.000,E1 292.770} C_DIS
LIN {X 0.235,Y -677.460,Z 966.424,A 0.000,B 0.000,C 90.000,E1 292.280} C_DIS
LIN {X -0.211,Y -677.405,Z 966.423,A 0.000,B 0.000,C 90.000,E1 292.078} C_DIS
LIN {X -0.101,Y -676.870,Z 966.420,A 0.000,B 0.000,C 90.000,E1 291.589} C_DIS
LIN {X -0.170,Y -676.148,Z 966.419,A 0.000,B 0.000,C 90.000,E1 291.354} C_DIS
LIN {X -0.063,Y -673.639,Z 966.416,A 0.000,B 0.000,C 90.000,E1 290.865} C_DIS
LIN {X 0.020,Y -672.860,Z 966.415,A 0.000,B 0.000,C 90.000,E1 290.737} C_DIS
LIN {X 0.102,Y -671.703,Z 966.415,A 0.000,B 0.000,C 90.000,E1 290.610} C_DIS
LIN {X 0.025,Y -665.742,Z 966.412,A 0.000,B 0.000,C 90.000,E1 290.174} C_DIS
LIN {X -0.034,Y -657.922,Z 966.409,A 0.000,B 0.000,C 90.000,E1 289.685} C_DIS
LIN {X 0.052,Y -655.810,Z 966.409,A 0.000,B 0.000,C 90.000,E1 289.523} C_DIS
LIN {X 0.236,Y -655.776,Z 966.409,A 0.000,B 0.000,C 90.000,E1 289.504} C_DIS
LIN {X 0.114,Y -655.114,Z 966.408,A 0.000,B 0.000,C 90.000,E1 289.396} C_DIS
LIN {X 0.077,Y -655.111,Z 966.408,A 0.000,B 0.000,C 90.000,E1 289.396} C_DIS
LIN {X -0.052,Y -655.374,Z 966.406,A 0.000,B 0.000,C 90.000,E1 289.141} C_DIS
LIN {X -0.089,Y -657.393,Z 966.404,A 0.000,B 0.000,C 90.000,E1 288.652} C_DIS
LIN {X 0.151,Y -663.972,Z 966.398,A 0.000,B 0.000,C 90.000,E1 287.528} C_DIS
LIN {X 0.223,Y -667.288,Z 966.394,A 0.000,B 0.000,C 90.000,E1 286.913} C_DIS
LIN {X 0.141,Y -668.556,Z 966.393,A 0.000,B 0.000,C 90.000,E1 286.677} C_DIS
LIN {X -0.081,Y -671.681,Z 966.389,A 0.000,B 0.000,C 90.000,E1 285.969} C_DIS
LIN {X -0.031,Y -673.292,Z 966.386,A 0.000,B 0.000,C 90.000,E1 285.481} C_DIS
LIN {X -0.207,Y -675.307,Z 966.382,A 0.000,B 0.000,C 90.000,E1 284.773} C_DIS
LIN {X 0.293,Y -676.756,Z 966.378,A 0.000,B 0.000,C 90.000,E1 284.008} C_DIS
LIN {X 0.110,Y -678.173,Z 966.373,A 0.000,B 0.000,C 90.000,E1 283.063} C_DIS
LIN {X -0.021,Y -678.860,Z 966.369,A 0.000,B 0.000,C 90.000,E1 282.355} C_DIS
LIN {X -0.107,Y -679.150,Z 966.366,A 0.000,B 0.000,C 90.000,E1 281.883} C_DIS
LIN {X -0.328,Y -679.222,Z 966.363,A 0.000,B 0.000,C 90.000,E1 281.422} C_DIS
LIN {X 0.209,Y -678.872,Z 966.359,A 0.000,B 0.000,C 90.000,E1 280.658} C_DIS
LIN {X -0.006,Y -678.370,Z 966.357,A 0.000,B 0.000,C 90.000,E1 280.197} C_DIS
LIN {X -0.102,Y -677.546,Z 966.354,A 0.000,B 0.000,C 90.000,E1 279.726} C_DIS
LIN {X -0.320,Y -676.513,Z 966.351,A 0.000,B 0.000,C 90.000,E1 279.265} C_DIS
LIN {X 0.128,Y -675.136,Z 966.349,A 0.000,B 0.000,C 90.000,E1 278.746} C_DIS
LIN {X 0.066,Y -674.344,Z 966.347,A 0.000,B 0.000,C 90.000,E1 278.511} C_DIS
LIN {X -0.237,Y -671.489,Z 966.343,A 0.000,B 0.000,C 90.000,E1 277.814} C_DIS
LIN {X 0.261,Y -670.475,Z 966.342,A 0.000,B 0.000,C 90.000,E1 277.530} C_DIS
LIN {X -0.084,Y -666.675,Z 966.338,A 0.000,B 0.000,C 90.000,E1 276.834} C_DIS
LIN {X 0.297,Y -663.760,Z 966.335,A 0.000,B 0.000,C 90.000,E1 276.315} C_DIS
LIN {X -0.002,Y -660.469,Z 966.333,A 0.000,B 0.000,C 90.000,E1 275.853} C_DIS
LIN {X 0.232,Y -655.698,Z 966.329,A 0.000,B 0.000,C 90.000,E1 275.220} C_DIS
LIN {X -0.119,Y -651.460,Z 966.326,A 0.000,B 0.000,C 90.000,E1 274.759} C_DIS
LIN {X -0.008,Y -645.703,Z 966.323,A 0.000,B 0.000,C 90.000,E1 274.131} C_DIS
LIN {X -0.189,Y -640.949,Z 966.320,A 0.000,B 0.000,C 90.000,E1 273.669} C_DIS
LIN {X 0.203,Y -635.736,Z 966.318,A 0.000,B 0.000,C 90.000,E1 273.154} C_DIS
LIN {X 0.277,Y -630.311,Z 966.315,A 0.000,B 0.000,C 90.000,E1 272.694} C_DIS
LIN {X -0.153,Y -624.701,Z 966.313,A 0.000,B 0.000,C 90.000,E1 272.293} C_DIS
LIN {X 0.189,Y -618.740,Z 966.310,A 0.000,B 0.000,C 90.000,E1 271.835} C_DIS
LIN {X -0.172,Y -610.955,Z 966.308,A 0.000,B 0.000,C 90.000,E1 271.375} C_DIS
LIN {X 0.211,Y -604.474,Z 966.306,A 0.000,B 0.000,C 90.000,E1 270.974} C_DIS
LIN {X -0.282,Y -597.700,Z 966.304,A 0.000,B 0.000,C 90.000,E1 270.688} C_DIS
LIN {X 0.263,Y -590.751,Z 966.302,A 0.000,B 0.000,C 90.000,E1 270.344} C_DIS
LIN {X -0.015,Y -585.513,Z 966.301,A 0.000,B 0.000,C 90.000,E1 270.172} C_DIS
LIN {X -0.120,Y -578.006,Z 966.300,A 0.000,B 0.000,C 90.000,E1 269.943} C_DIS
LIN {X 0.035,Y -572.045,Z 966.299,A 0.000,B 0.000,C 90.000,E1 269.771} C_DIS
LIN {X -0.102,Y -565.986,Z 966.298,A 0.000,B 0.000,C 90.000,E1 269.656} C_DIS
LIN {X -0.245,Y -560.893,Z 966.298,A 0.000,B 0.000,C 90.000,E1 269.599} C_DIS
LIN {X -0.089,Y -557.236,Z 966.297,A 0.000,B 0.000,C 90.000,E1 269.542} C_DIS
LIN {X -0.146,Y -552.113,Z 966.297,A 0.000,B 0.000,C 90.000,E1 269.542} C_DIS
LIN {X -0.193,Y -547.053,Z 966.297,A 0.000,B 0.000,C 90.000,E1 269.542} C_DIS
LIN {X 0.127,Y -543.096,Z 966.296,A 0.000,B 0.000,C 90.000,E1 269.312} C_DIS
LIN {X 0.079,Y -543.016,Z 966.296,A 0.000,B 0.000,C 90.000,E1 269.312} C_DIS
LIN {X 0.061,Y -542.666,Z 966.295,A 0.000,B 0.000,C 90.000,E1 269.026} C_DIS
LIN {X -0.140,Y -542.146,Z 966.291,A 0.000,B 0.000,C 90.000,E1 268.339} C_DIS
LIN {X 0.135,Y -540.298,Z 966.277,A 0.000,B 0.000,C 90.000,E1 265.755} C_DIS
LIN {X -0.258,Y -539.291,Z 966.269,A 0.000,B 0.000,C 90.000,E1 264.375} C_DIS
LIN {X -0.136,Y -538.473,Z 966.262,A 0.000,B 0.000,C 90.000,E1 263.223} C_DIS
LIN {X 0.022,Y -537.225,Z 966.254,A 0.000,B 0.000,C 90.000,E1 261.781} C_DIS
LIN {X 0.231,Y -535.738,Z 966.246,A 0.000,B 0.000,C 90.000,E1 260.330} C_DIS
LIN {X -0.070,Y -534.468,Z 966.240,A 0.000,B 0.000,C 90.000,E1 259.218} C_DIS
LIN {X -0.237,Y -532.077,Z 966.229,A 0.000,B 0.000,C 90.000,E1 257.229} C_DIS
LIN {X -0.188,Y -529.307,Z 966.216,A 0.000,B 0.000,C 90.000,E1 254.921} C_DIS
LIN {X 0.076,Y -527.794,Z 966.208,A 0.000,B 0.000,C 90.000,E1 253.449} C_DIS
LIN {X 0.099,Y -526.173,Z 966.200,A 0.000,B 0.000,C 90.000,E1 252.000} C_DIS
LIN {X 0.260,Y -523.940,Z 966.190,A 0.000,B 0.000,C 90.000,E1 250.242} C_DIS
LIN {X 0.234,Y -522.442,Z 966.184,A 0.000,B 0.000,C 90.000,E1 249.082} C_DIS
LIN {X 0.002,Y -520.217,Z 966.174,A 0.000,B 0.000,C 90.000,E1 247.358} C_DIS
LIN {X -0.084,Y -517.628,Z 966.164,A 0.000,B 0.000,C 90.000,E1 245.613} C_DIS
LIN {X 0.195,Y -515.807,Z 966.158,A 0.000,B 0.000,C 90.000,E1 244.409} C_DIS
LIN {X -0.010,Y -513.084,Z 966.148,A 0.000,B 0.000,C 90.000,E1 242.666} C_DIS
LIN {X 0.082,Y -510.668,Z 966.140,A 0.000,B 0.000,C 90.000,E1 241.179} C_DIS
LIN {X 0.038,Y -508.651,Z 966.133,A 0.000,B 0.000,C 90.000,E1 239.999} C_DIS
LIN {X -0.043,Y -506.408,Z 966.127,A 0.000,B 0.000,C 90.000,E1 238.820} C_DIS
LIN {X -0.328,Y -504.034,Z 966.120,A 0.000,B 0.000,C 90.000,E1 237.661} C_DIS
LIN {X 0.054,Y -501.452,Z 966.114,A 0.000,B 0.000,C 90.000,E1 236.421} C_DIS
LIN {X 0.139,Y -497.302,Z 966.104,A 0.000,B 0.000,C 90.000,E1 234.609} C_DIS
LIN {X -0.274,Y -493.293,Z 966.093,A 0.000,B 0.000,C 90.000,E1 232.844} C_DIS
LIN {X -0.179,Y -489.078,Z 966.083,A 0.000,B 0.000,C 90.000,E1 231.009} C_DIS
LIN {X -0.046,Y -484.094,Z 966.071,A 0.000,B 0.000,C 90.000,E1 228.852} C_DIS
LIN {X 0.101,Y -479.870,Z 966.061,A 0.000,B 0.000,C 90.000,E1 226.986} C_DIS
LIN {X -0.194,Y -475.838,Z 966.051,A 0.000,B 0.000,C 90.000,E1 225.162} C_DIS
LIN {X -0.004,Y -472.364,Z 966.042,A 0.000,B 0.000,C 90.000,E1 223.581} C_DIS
LIN {X 0.271,Y -470.314,Z 966.037,A 0.000,B 0.000,C 90.000,E1 222.609} C_DIS
LIN {X 0.032,Y -466.827,Z 966.028,A 0.000,B 0.000,C 90.000,E1 221.067} C_DIS
LIN {X 0.075,Y -463.399,Z 966.019,A 0.000,B 0.000,C 90.000,E1 219.483} C_DIS
LIN {X -0.013,Y -457.731,Z 966.005,A 0.000,B 0.000,C 90.000,E1 216.950} C_DIS
LIN {X 0.012,Y -453.410,Z 965.995,A 0.000,B 0.000,C 90.000,E1 215.025} C_DIS
LIN {X 0.043,Y -449.179,Z 965.984,A 0.000,B 0.000,C 90.000,E1 213.086} C_DIS
LIN {X 0.172,Y -444.328,Z 965.971,A 0.000,B 0.000,C 90.000,E1 210.797} C_DIS
LIN {X -0.066,Y -439.318,Z 965.959,A 0.000,B 0.000,C 90.000,E1 208.537} C_DIS
LIN {X 0.091,Y -435.010,Z 965.948,A 0.000,B 0.000,C 90.000,E1 206.539} C_DIS
LIN {X 0.141,Y -432.060,Z 965.940,A 0.000,B 0.000,C 90.000,E1 205.207} C_DIS
LIN {X -0.032,Y -428.963,Z 965.933,A 0.000,B 0.000,C 90.000,E1 203.898} C_DIS
LIN {X 0.067,Y -422.187,Z 965.916,A 0.000,B 0.000,C 90.000,E1 200.865} C_DIS
LIN {X -0.236,Y -418.639,Z 965.907,A 0.000,B 0.000,C 90.000,E1 199.214} C_DIS
LIN {X -0.046,Y -413.843,Z 965.893,A 0.000,B 0.000,C 90.000,E1 196.804} C_DIS
LIN {X 0.131,Y -410.577,Z 965.884,A 0.000,B 0.000,C 90.000,E1 195.064} C_DIS
LIN {X 0.024,Y -407.195,Z 965.874,A 0.000,B 0.000,C 90.000,E1 193.355} C_DIS
LIN {X 0.156,Y -404.499,Z 965.867,A 0.000,B 0.000,C 90.000,E1 191.951} C_DIS
LIN {X -0.158,Y -400.532,Z 965.855,A 0.000,B 0.000,C 90.000,E1 189.905} C_DIS
LIN {X 0.144,Y -396.479,Z 965.843,A 0.000,B 0.000,C 90.000,E1 187.757} C_DIS
LIN {X -0.030,Y -390.575,Z 965.824,A 0.000,B 0.000,C 90.000,E1 184.245} C_DIS
LIN {X 0.123,Y -389.352,Z 965.818,A 0.000,B 0.000,C 90.000,E1 183.154} C_DIS
LIN {X -0.036,Y -388.970,Z 965.814,A 0.000,B 0.000,C 90.000,E1 182.465} C_DIS
LIN {X 0.139,Y -389.172,Z 965.809,A 0.000,B 0.000,C 90.000,E1 181.547} C_DIS
LIN {X 0.004,Y -389.820,Z 965.806,A 0.000,B 0.000,C 90.000,E1 181.031} C_DIS
LIN {X -0.039,Y -389.940,Z 965.805,A 0.000,B 0.000,C 90.000,E1 180.859} C_DIS
LIN {X 0.190,Y -391.196,Z 965.802,A 0.000,B 0.000,C 90.000,E1 180.344} C_DIS
LIN {X 0.028,Y -394.084,Z 965.798,A 0.000,B 0.000,C 90.000,E1 179.656} C_DIS
LIN {X -0.008,Y -394.905,Z 965.797,A 0.000,B 0.000,C 90.000,E1 179.484} C_DIS
LIN {X -0.010,Y -398.142,Z 965.794,A 0.000,B 0.000,C 90.000,E1 178.969} C_DIS
LIN {X -0.069,Y -400.958,Z 965.792,A 0.000,B 0.000,C 90.000,E1 178.625} C_DIS
LIN {X 0.112,Y -405.237,Z 965.790,A 0.000,B 0.000,C 90.000,E1 178.108} C_DIS
LIN {X 0.113,Y -413.903,Z 965.785,A 0.000,B 0.000,C 90.000,E1 177.306} C_DIS
LIN {X 0.057,Y -422.966,Z 965.781,A 0.000,B 0.000,C 90.000,E1 176.502} C_DIS
LIN {X -0.081,Y -432.014,Z 965.776,A 0.000,B 0.000,C 90.000,E1 175.698} C_DIS
LIN {X 0.201,Y -440.959,Z 965.771,A 0.000,B 0.000,C 90.000,E1 174.837} C_DIS
LIN {X 0.141,Y -451.252,Z 965.766,A 0.000,B 0.000,C 90.000,E1 173.856} C_DIS
LIN {X -0.053,Y -458.294,Z 965.762,A 0.000,B 0.000,C 90.000,E1 173.166} C_DIS
LIN {X 0.028,Y -465.158,Z 965.758,A 0.000,B 0.000,C 90.000,E1 172.413} C_DIS
LIN {X 0.191,Y -473.241,Z 965.753,A 0.000,B 0.000,C 90.000,E1 171.489} C_DIS
LIN {X 0.003,Y -478.514,Z 965.750,A 0.000,B 0.000,C 90.000,E1 170.905} C_DIS
LIN {X -0.173,Y -488.440,Z 965.743,A 0.000,B 0.000,C 90.000,E1 169.690} C_DIS
LIN {X -0.122,Y -497.752,Z 965.736,A 0.000,B 0.000,C 90.000,E1 168.465} C_DIS
LIN {X 0.240,Y -504.264,Z 965.731,A 0.000,B 0.000,C 90.000,E1 167.521} C_DIS
LIN {X -0.089,Y -511.522,Z 965.725,A 0.000,B 0.000,C 90.000,E1 166.520} C_DIS
LIN {X 0.151,Y -520.041,Z 965.718,A 0.000,B 0.000,C 90.000,E1 165.172} C_DIS
LIN {X 0.093,Y -524.628,Z 965.714,A 0.000,B 0.000,C 90.000,E1 164.448} C_DIS
LIN {X -0.047,Y -530.934,Z 965.708,A 0.000,B 0.000,C 90.000,E1 163.449} C_DIS
LIN {X -0.121,Y -537.964,Z 965.702,A 0.000,B 0.000,C 90.000,E1 162.308} C_DIS
LIN {X 0.009,Y -547.233,Z 965.693,A 0.000,B 0.000,C 90.000,E1 160.732} C_DIS
LIN {X 0.237,Y -554.633,Z 965.686,A 0.000,B 0.000,C 90.000,E1 159.444} C_DIS
LIN {X 0.178,Y -560.953,Z 965.680,A 0.000,B 0.000,C 90.000,E1 158.337} C_DIS
LIN {X 0.109,Y -567.568,Z 965.673,A 0.000,B 0.000,C 90.000,E1 157.102} C_DIS
LIN {X 0.357,Y -569.718,Z 965.671,A 0.000,B 0.000,C 90.000,E1 156.666} C_DIS
LIN {X -0.268,Y -577.083,Z 965.662,A 0.000,B 0.000,C 90.000,E1 155.229} C_DIS
LIN {X -0.256,Y -581.328,Z 965.657,A 0.000,B 0.000,C 90.000,E1 154.280} C_DIS
LIN {X -0.003,Y -585.837,Z 965.651,A 0.000,B 0.000,C 90.000,E1 153.179} C_DIS
LIN {X 0.162,Y -589.027,Z 965.647,A 0.000,B 0.000,C 90.000,E1 152.359} C_DIS
LIN {X 0.008,Y -592.745,Z 965.641,A 0.000,B 0.000,C 90.000,E1 151.307} C_DIS
LIN {X -0.183,Y -597.194,Z 965.633,A 0.000,B 0.000,C 90.000,E1 149.999} C_DIS
LIN {X -0.002,Y -601.499,Z 965.626,A 0.000,B 0.000,C 90.000,E1 148.663} C_DIS
LIN {X 0.327,Y -604.939,Z 965.620,A 0.000,B 0.000,C 90.000,E1 147.582} C_DIS
LIN {X -0.328,Y -606.608,Z 965.617,A 0.000,B 0.000,C 90.000,E1 147.120} C_DIS
LIN {X 0.128,Y -609.033,Z 965.613,A 0.000,B 0.000,C 90.000,E1 146.294} C_DIS
LIN {X 0.046,Y -612.431,Z 965.607,A 0.000,B 0.000,C 90.000,E1 145.261} C_DIS
LIN {X 0.108,Y -617.422,Z 965.598,A 0.000,B 0.000,C 90.000,E1 143.703} C_DIS
LIN {X -0.223,Y -622.270,Z 965.590,A 0.000,B 0.000,C 90.000,E1 142.190} C_DIS
LIN {X 0.075,Y -626.345,Z 965.583,A 0.000,B 0.000,C 90.000,E1 140.884} C_DIS
LIN {X -0.176,Y -631.081,Z 965.574,A 0.000,B 0.000,C 90.000,E1 139.380} C_DIS
LIN {X 0.088,Y -635.952,Z 965.566,A 0.000,B 0.000,C 90.000,E1 137.838} C_DIS
LIN {X 0.077,Y -640.158,Z 965.559,A 0.000,B 0.000,C 90.000,E1 136.581} C_DIS
LIN {X -0.011,Y -646.071,Z 965.549,A 0.000,B 0.000,C 90.000,E1 134.838} C_DIS
LIN {X -0.061,Y -653.903,Z 965.537,A 0.000,B 0.000,C 90.000,E1 132.609} C_DIS
LIN {X 0.154,Y -662.072,Z 965.524,A 0.000,B 0.000,C 90.000,E1 130.378} C_DIS
LIN {X 0.141,Y -665.761,Z 965.519,A 0.000,B 0.000,C 90.000,E1 129.402} C_DIS
LIN {X 0.186,Y -668.460,Z 965.515,A 0.000,B 0.000,C 90.000,E1 128.669} C_DIS
LIN {X -0.057,Y -673.600,Z 965.507,A 0.000,B 0.000,C 90.000,E1 127.237} C_DIS
LIN {X -0.342,Y -676.827,Z 965.502,A 0.000,B 0.000,C 90.000,E1 126.297} C_DIS
LIN {X -0.042,Y -679.881,Z 965.496,A 0.000,B 0.000,C 90.000,E1 125.311} C_DIS
LIN {X 0.298,Y -682.812,Z 965.491,A 0.000,B 0.000,C 90.000,E1 124.326} C_DIS
LIN {X 0.293,Y -685.500,Z 965.486,A 0.000,B 0.000,C 90.000,E1 123.372} C_DIS
LIN {X 0.173,Y -689.275,Z 965.478,A 0.000,B 0.000,C 90.000,E1 121.957} C_DIS
LIN {X 0.255,Y -691.590,Z 965.472,A 0.000,B 0.000,C 90.000,E1 121.003} C_DIS
LIN {X 0.006,Y -693.695,Z 965.467,A 0.000,B 0.000,C 90.000,E1 120.079} C_DIS
LIN {X 0.141,Y -695.089,Z 965.463,A 0.000,B 0.000,C 90.000,E1 119.361} C_DIS
LIN {X -0.063,Y -696.390,Z 965.458,A 0.000,B 0.000,C 90.000,E1 118.437} C_DIS
LIN {X 0.000,Y -697.710,Z 965.451,A 0.000,B 0.000,C 90.000,E1 117.257} C_DIS
LIN {X 0.120,Y -698.485,Z 965.446,A 0.000,B 0.000,C 90.000,E1 116.309} C_DIS
LIN {X -0.107,Y -699.106,Z 965.440,A 0.000,B 0.000,C 90.000,E1 115.155} C_DIS
LIN {X -0.232,Y -699.294,Z 965.436,A 0.000,B 0.000,C 90.000,E1 114.463} C_DIS
LIN {X 0.034,Y -699.244,Z 965.435,A 0.000,B 0.000,C 90.000,E1 114.207} C_DIS
LIN {X -0.357,Y -698.897,Z 965.432,A 0.000,B 0.000,C 90.000,E1 113.770} C_DIS
LIN {X 0.169,Y -697.774,Z 965.429,A 0.000,B 0.000,C 90.000,E1 113.259} C_DIS
LIN {X 0.154,Y -697.039,Z 965.428,A 0.000,B 0.000,C 90.000,E1 113.025} C_DIS
LIN {X 0.283,Y -696.408,Z 965.427,A 0.000,B 0.000,C 90.000,E1 112.898} C_DIS
LIN {X -0.124,Y -692.715,Z 965.425,A 0.000,B 0.000,C 90.000,E1 112.461} C_DIS
LIN {X -0.003,Y -691.615,Z 965.424,A 0.000,B 0.000,C 90.000,E1 112.333} C_DIS
LIN {X 0.115,Y -689.950,Z 965.423,A 0.000,B 0.000,C 90.000,E1 112.206} C_DIS
LIN {X -0.015,Y -685.704,Z 965.422,A 0.000,B 0.000,C 90.000,E1 112.025} C_DIS
LIN {X -0.201,Y -680.060,Z 965.421,A 0.000,B 0.000,C 90.000,E1 111.844} C_DIS
LIN {X 0.003,Y -675.755,Z 965.421,A 0.000,B 0.000,C 90.000,E1 111.716} C_DIS
LIN {X -0.363,Y -670.570,Z 965.421,A 0.000,B 0.000,C 90.000,E1 111.716} C_DIS
LIN {X 0.141,Y -668.015,Z 965.420,A 0.000,B 0.000,C 90.000,E1 111.663} C_DIS
LIN {X 0.087,Y -627.952,Z 965.420,A 0.000,B 0.000,C 90.000,E1 111.663} C_DIS
LIN {X -0.187,Y -621.872,Z 965.420,A 0.000,B 0.000,C 90.000,E1 111.589} C_DIS
LIN {X -0.216,Y -616.451,Z 965.419,A 0.000,B 0.000,C 90.000,E1 111.461} C_DIS
LIN {X -0.166,Y -609.421,Z 965.418,A 0.000,B 0.000,C 90.000,E1 111.227} C_DIS
LIN {X 0.177,Y -604.145,Z 965.417,A 0.000,B 0.000,C 90.000,E1 110.972} C_DIS
LIN {X 0.053,Y -598.091,Z 965.415,A 0.000,B 0.000,C 90.000,E1 110.663} C_DIS
LIN {X 0.233,Y -590.862,Z 965.412,A 0.000,B 0.000,C 90.000,E1 110.174} C_DIS
LIN {X -0.112,Y -574.867,Z 965.406,A 0.000,B 0.000,C 90.000,E1 109.014} C_DIS
LIN {X 0.093,Y -568.331,Z 965.403,A 0.000,B 0.000,C 90.000,E1 108.598} C_DIS
LIN {X 0.218,Y -561.275,Z 965.401,A 0.000,B 0.000,C 90.000,E1 108.236} C_DIS
LIN {X -0.067,Y -552.542,Z 965.399,A 0.000,B 0.000,C 90.000,E1 107.819} C_DIS
LIN {X -0.068,Y -550.588,Z 965.398,A 0.000,B 0.000,C 90.000,E1 107.638} C_DIS
LIN {X -0.106,Y -550.563,Z 965.398,A 0.000,B 0.000,C 90.000,E1 107.638} C_DIS
LIN {X -0.228,Y -550.092,Z 965.397,A 0.000,B 0.000,C 90.000,E1 107.457} C_DIS
LIN {X 0.128,Y -550.010,Z 965.394,A 0.000,B 0.000,C 90.000,E1 106.858} C_DIS
LIN {X 0.159,Y -550.536,Z 965.388,A 0.000,B 0.000,C 90.000,E1 105.733} C_DIS
LIN {X 0.075,Y -551.911,Z 965.372,A 0.000,B 0.000,C 90.000,E1 102.939} C_DIS
LIN {X 0.216,Y -554.468,Z 965.355,A 0.000,B 0.000,C 90.000,E1 99.849} C_DIS
LIN {X -0.207,Y -556.066,Z 965.346,A 0.000,B 0.000,C 90.000,E1 98.219} C_DIS
LIN {X 0.159,Y -557.102,Z 965.339,A 0.000,B 0.000,C 90.000,E1 97.068} C_DIS
LIN {X 0.124,Y -558.197,Z 965.332,A 0.000,B 0.000,C 90.000,E1 95.682} C_DIS
LIN {X -0.030,Y -558.997,Z 965.326,A 0.000,B 0.000,C 90.000,E1 94.588} C_DIS
LIN {X 0.076,Y -560.109,Z 965.315,A 0.000,B 0.000,C 90.000,E1 92.636} C_DIS
LIN {X 0.185,Y -561.129,Z 965.304,A 0.000,B 0.000,C 90.000,E1 90.688} C_DIS
LIN {X 0.111,Y -561.630,Z 965.296,A 0.000,B 0.000,C 90.000,E1 89.312} C_DIS
LIN {X 0.059,Y -561.986,Z 965.289,A 0.000,B 0.000,C 90.000,E1 87.936} C_DIS
LIN {X 0.112,Y -562.334,Z 965.279,A 0.000,B 0.000,C 90.000,E1 86.274} C_DIS
LIN {X -0.223,Y -562.589,Z 965.269,A 0.000,B 0.000,C 90.000,E1 84.375} C_DIS
LIN {X 0.246,Y -562.733,Z 965.263,A 0.000,B 0.000,C 90.000,E1 83.223} C_DIS
LIN {X -0.024,Y -563.128,Z 965.252,A 0.000,B 0.000,C 90.000,E1 81.319} C_DIS
LIN {X 0.211,Y -564.042,Z 965.238,A 0.000,B 0.000,C 90.000,E1 78.814} C_DIS
LIN {X 0.261,Y -565.028,Z 965.227,A 0.000,B 0.000,C 90.000,E1 76.881} C_DIS
LIN {X 0.128,Y -565.920,Z 965.220,A 0.000,B 0.000,C 90.000,E1 75.519} C_DIS
LIN {X -0.046,Y -567.235,Z 965.209,A 0.000,B 0.000,C 90.000,E1 73.614} C_DIS
LIN {X 0.019,Y -568.136,Z 965.201,A 0.000,B 0.000,C 90.000,E1 72.236} C_DIS
LIN {X -0.105,Y -569.116,Z 965.192,A 0.000,B 0.000,C 90.000,E1 70.604} C_DIS
LIN {X -0.020,Y -569.873,Z 965.183,A 0.000,B 0.000,C 90.000,E1 68.954} C_DIS
LIN {X 0.112,Y -570.348,Z 965.177,A 0.000,B 0.000,C 90.000,E1 67.847} C_DIS
LIN {X -0.100,Y -570.918,Z 965.168,A 0.000,B 0.000,C 90.000,E1 66.230} C_DIS
LIN {X -0.071,Y -571.316,Z 965.159,A 0.000,B 0.000,C 90.000,E1 64.588} C_DIS
LIN {X 0.124,Y -571.645,Z 965.151,A 0.000,B 0.000,C 90.000,E1 63.204} C_DIS
LIN {X 0.168,Y -571.880,Z 965.142,A 0.000,B 0.000,C 90.000,E1 61.563} C_DIS
LIN {X -0.057,Y -571.990,Z 965.133,A 0.000,B 0.000,C 90.000,E1 59.950} C_DIS
LIN {X -0.033,Y -572.167,Z 965.125,A 0.000,B 0.000,C 90.000,E1 58.584} C_DIS
LIN {X -0.298,Y -572.241,Z 965.118,A 0.000,B 0.000,C 90.000,E1 57.248} C_DIS
LIN {X -0.262,Y -572.071,Z 965.110,A 0.000,B 0.000,C 90.000,E1 55.881} C_DIS
LIN {X 0.091,Y -571.806,Z 965.103,A 0.000,B 0.000,C 90.000,E1 54.482} C_DIS
LIN {X 0.365,Y -571.670,Z 965.100,A 0.000,B 0.000,C 90.000,E1 53.909} C_DIS
LIN {X 0.111,Y -571.119,Z 965.094,A 0.000,B 0.000,C 90.000,E1 52.844} C_DIS
LIN {X 0.063,Y -570.599,Z 965.089,A 0.000,B 0.000,C 90.000,E1 52.029} C_DIS
LIN {X -0.342,Y -569.969,Z 965.085,A 0.000,B 0.000,C 90.000,E1 51.251} C_DIS
LIN {X 0.212,Y -568.670,Z 965.077,A 0.000,B 0.000,C 90.000,E1 49.828} C_DIS
LIN {X -0.175,Y -567.316,Z 965.071,A 0.000,B 0.000,C 90.000,E1 48.771} C_DIS
LIN {X 0.111,Y -566.104,Z 965.066,A 0.000,B 0.000,C 90.000,E1 47.919} C_DIS
LIN {X -0.099,Y -565.227,Z 965.063,A 0.000,B 0.000,C 90.000,E1 47.391} C_DIS
LIN {X -0.159,Y -563.126,Z 965.057,A 0.000,B 0.000,C 90.000,E1 46.296} C_DIS
LIN {X -0.005,Y -561.963,Z 965.054,A 0.000,B 0.000,C 90.000,E1 45.729} C_DIS
LIN {X -0.184,Y -560.015,Z 965.049,A 0.000,B 0.000,C 90.000,E1 44.919} C_DIS
LIN {X -0.051,Y -558.626,Z 965.046,A 0.000,B 0.000,C 90.000,E1 44.352} C_DIS
LIN {X 0.177,Y -555.284,Z 965.040,A 0.000,B 0.000,C 90.000,E1 43.218} C_DIS
LIN {X -0.107,Y -553.421,Z 965.037,A 0.000,B 0.000,C 90.000,E1 42.690} C_DIS
LIN {X -0.028,Y -551.433,Z 965.034,A 0.000,B 0.000,C 90.000,E1 42.123} C_DIS
LIN {X -0.284,Y -548.185,Z 965.029,A 0.000,B 0.000,C 90.000,E1 41.310} C_DIS
LIN {X -0.035,Y -546.428,Z 965.027,A 0.000,B 0.000,C 90.000,E1 40.862} C_DIS
LIN {X -0.178,Y -543.166,Z 965.023,A 0.000,B 0.000,C 90.000,E1 40.172} C_DIS
LIN {X 0.039,Y -541.201,Z 965.021,A 0.000,B 0.000,C 90.000,E1 39.725} C_DIS
LIN {X 0.024,Y -535.244,Z 965.014,A 0.000,B 0.000,C 90.000,E1 38.588} C_DIS
LIN {X 0.018,Y -530.331,Z 965.010,A 0.000,B 0.000,C 90.000,E1 37.729} C_DIS
LIN {X -0.039,Y -525.243,Z 965.005,A 0.000,B 0.000,C 90.000,E1 36.870} C_DIS
LIN {X 0.028,Y -520.771,Z 965.001,A 0.000,B 0.000,C 90.000,E1 36.137} C_DIS
LIN {X 0.284,Y -515.144,Z 964.996,A 0.000,B 0.000,C 90.000,E1 35.231} C_DIS
LIN {X -0.049,Y -510.151,Z 964.992,A 0.000,B 0.000,C 90.000,E1 34.532} C_DIS
LIN {X 0.000,Y -504.609,Z 964.988,A 0.000,B 0.000,C 90.000,E1 33.785} C_DIS
LIN {X -0.302,Y -501.151,Z 964.985,A 0.000,B 0.000,C 90.000,E1 33.372} C_DIS
LIN {X -0.111,Y -495.189,Z 964.981,A 0.000,B 0.000,C 90.000,E1 32.625} C_DIS
LIN {X 0.255,Y -491.114,Z 964.979,A 0.000,B 0.000,C 90.000,E1 32.133} C_DIS
LIN {X 0.284,Y -482.883,Z 964.974,A 0.000,B 0.000,C 90.000,E1 31.258} C_DIS
LIN {X -0.012,Y -475.637,Z 964.970,A 0.000,B 0.000,C 90.000,E1 30.590} C_DIS
LIN {X 0.180,Y -466.934,Z 964.965,A 0.000,B 0.000,C 90.000,E1 29.745} C_DIS
LIN {X 0.088,Y -457.985,Z 964.961,A 0.000,B 0.000,C 90.000,E1 28.949} C_DIS
LIN {X 0.098,Y -450.321,Z 964.957,A 0.000,B 0.000,C 90.000,E1 28.281} C_DIS
LIN {X 0.027,Y -438.187,Z 964.951,A 0.000,B 0.000,C 90.000,E1 27.257} C_DIS
LIN {X 0.266,Y -415.677,Z 964.940,A 0.000,B 0.000,C 90.000,E1 25.207} C_DIS
LIN {X 0.135,Y -402.451,Z 964.933,A 0.000,B 0.000,C 90.000,E1 23.898} C_DIS
LIN {X -0.207,Y -397.051,Z 964.930,A 0.000,B 0.000,C 90.000,E1 23.334} C_DIS
LIN {X -0.111,Y -394.624,Z 964.928,A 0.000,B 0.000,C 90.000,E1 23.003} C_DIS
LIN {X -0.016,Y -392.852,Z 964.926,A 0.000,B 0.000,C 90.000,E1 22.642} C_DIS
LIN {X 0.011,Y -391.792,Z 964.925,A 0.000,B 0.000,C 90.000,E1 22.461} C_DIS
LIN {X 0.227,Y -390.178,Z 964.922,A 0.000,B 0.000,C 90.000,E1 21.897} C_DIS
LIN {X -0.058,Y -389.649,Z 964.918,A 0.000,B 0.000,C 90.000,E1 21.227} C_DIS
LIN {X 0.175,Y -389.869,Z 964.913,A 0.000,B 0.000,C 90.000,E1 20.301} C_DIS
LIN {X -0.129,Y -394.821,Z 964.885,A 0.000,B 0.000,C 90.000,E1 15.371} C_DIS
LIN {X -0.071,Y -397.481,Z 964.874,A 0.000,B 0.000,C 90.000,E1 13.244} C_DIS
LIN {X 0.001,Y -402.170,Z 964.856,A 0.000,B 0.000,C 90.000,E1 10.074} C_DIS
LIN {X -0.044,Y -407.681,Z 964.839,A 0.000,B 0.000,C 90.000,E1 6.947} C_DIS
LIN {X -0.052,Y -411.017,Z 964.829,A 0.000,B 0.000,C 90.000,E1 5.220} C_DIS
LIN {X 0.012,Y -416.086,Z 964.816,A 0.000,B 0.000,C 90.000,E1 2.808} C_DIS
LIN {X 0.122,Y -419.896,Z 964.806,A 0.000,B 0.000,C 90.000,E1 1.088} C_DIS
LIN {X 0.185,Y -421.523,Z 964.802,A 0.000,B 0.000,C 90.000,E1 0.401} C_DIS
LIN {X 0.000,Y -422.701,Z 964.800,A 0.000,B 0.000,C 90.000,E1 360.000} C_DIS
LIN {X -0.173,Y -425.150,Z 964.796,A 0.000,B 0.000,C 90.000,E1 359.370} C_DIS
LIN {X 0.199,Y -428.200,Z 964.794,A 0.000,B 0.000,C 90.000,E1 358.797} C_DIS
LIN {X -0.200,Y -429.418,Z 964.793,A 0.000,B 0.000,C 90.000,E1 358.682} C_DIS
LIN {X 0.181,Y -434.591,Z 964.790,A 0.000,B 0.000,C 90.000,E1 358.167} C_DIS
LIN {X -0.019,Y -440.656,Z 964.788,A 0.000,B 0.000,C 90.000,E1 357.822} C_DIS
LIN {X 0.056,Y -446.068,Z 964.786,A 0.000,B 0.000,C 90.000,E1 357.535} C_DIS
LIN {X -0.085,Y -464.520,Z 964.781,A 0.000,B 0.000,C 90.000,E1 356.560} C_DIS
LIN {X 0.020,Y -472.904,Z 964.778,A 0.000,B 0.000,C 90.000,E1 356.102} C_DIS
LIN {X -0.103,Y -484.529,Z 964.775,A 0.000,B 0.000,C 90.000,E1 355.469} C_DIS
LIN {X -0.048,Y -495.712,Z 964.771,A 0.000,B 0.000,C 90.000,E1 354.837} C_DIS
LIN {X 0.092,Y -505.384,Z 964.768,A 0.000,B 0.000,C 90.000,E1 354.261} C_DIS
LIN {X 0.061,Y -516.309,Z 964.764,A 0.000,B 0.000,C 90.000,E1 353.571} C_DIS
LIN {X 0.268,Y -525.561,Z 964.761,A 0.000,B 0.000,C 90.000,E1 352.932} C_DIS
LIN {X -0.031,Y -533.007,Z 964.758,A 0.000,B 0.000,C 90.000,E1 352.413} C_DIS
LIN {X -0.167,Y -540.137,Z 964.755,A 0.000,B 0.000,C 90.000,E1 351.837} C_DIS
LIN {X 0.033,Y -547.002,Z 964.751,A 0.000,B 0.000,C 90.000,E1 351.197} C_DIS
LIN {X 0.005,Y -554.527,Z 964.747,A 0.000,B 0.000,C 90.000,E1 350.443} C_DIS
LIN {X 0.088,Y -558.210,Z 964.745,A 0.000,B 0.000,C 90.000,E1 350.038} C_DIS
LIN {X 0.214,Y -563.802,Z 964.741,A 0.000,B 0.000,C 90.000,E1 349.342} C_DIS
LIN {X 0.157,Y -567.909,Z 964.738,A 0.000,B 0.000,C 90.000,E1 348.814} C_DIS
LIN {X -0.041,Y -571.825,Z 964.735,A 0.000,B 0.000,C 90.000,E1 348.285} C_DIS
LIN {X -0.008,Y -577.270,Z 964.730,A 0.000,B 0.000,C 90.000,E1 347.465} C_DIS
LIN {X 0.185,Y -581.386,Z 964.727,A 0.000,B 0.000,C 90.000,E1 346.769} C_DIS
LIN {X -0.117,Y -586.066,Z 964.722,A 0.000,B 0.000,C 90.000,E1 345.992} C_DIS
LIN {X -0.257,Y -591.865,Z 964.716,A 0.000,B 0.000,C 90.000,E1 344.936} C_DIS
LIN {X -0.172,Y -597.249,Z 964.710,A 0.000,B 0.000,C 90.000,E1 343.866} C_DIS
LIN {X -0.070,Y -602.874,Z 964.704,A 0.000,B 0.000,C 90.000,E1 342.670} C_DIS
LIN {X -0.236,Y -607.521,Z 964.698,A 0.000,B 0.000,C 90.000,E1 341.638} C_DIS
LIN {X 0.242,Y -611.907,Z 964.692,A 0.000,B 0.000,C 90.000,E1 340.550} C_DIS
LIN {X 0.202,Y -616.067,Z 964.686,A 0.000,B 0.000,C 90.000,E1 339.518} C_DIS
LIN {X -0.117,Y -618.989,Z 964.682,A 0.000,B 0.000,C 90.000,E1 338.773} C_DIS
LIN {X 0.163,Y -622.621,Z 964.676,A 0.000,B 0.000,C 90.000,E1 337.720} C_DIS
LIN {X -0.320,Y -626.822,Z 964.669,A 0.000,B 0.000,C 90.000,E1 336.485} C_DIS
LIN {X 0.080,Y -630.836,Z 964.662,A 0.000,B 0.000,C 90.000,E1 335.177} C_DIS
LIN {X 0.242,Y -634.398,Z 964.655,A 0.000,B 0.000,C 90.000,E1 333.896} C_DIS
LIN {X -0.147,Y -636.952,Z 964.650,A 0.000,B 0.000,C 90.000,E1 332.922} C_DIS
LIN {X 0.065,Y -639.344,Z 964.644,A 0.000,B 0.000,C 90.000,E1 331.897} C_DIS
LIN {X 0.181,Y -642.699,Z 964.636,A 0.000,B 0.000,C 90.000,E1 330.383} C_DIS
LIN {X -0.107,Y -644.749,Z 964.630,A 0.000,B 0.000,C 90.000,E1 329.410} C_DIS
LIN {X -0.048,Y -646.493,Z 964.625,A 0.000,B 0.000,C 90.000,E1 328.408} C_DIS
LIN {X -0.095,Y -648.518,Z 964.618,A 0.000,B 0.000,C 90.000,E1 327.168} C_DIS
LIN {X -0.099,Y -650.141,Z 964.611,A 0.000,B 0.000,C 90.000,E1 325.928} C_DIS
LIN {X -0.083,Y -651.575,Z 964.604,A 0.000,B 0.000,C 90.000,E1 324.689} C_DIS
LIN {X -0.120,Y -652.487,Z 964.598,A 0.000,B 0.000,C 90.000,E1 323.703} C_DIS
LIN {X -0.218,Y -653.397,Z 964.591,A 0.000,B 0.000,C 90.000,E1 322.477} C_DIS
LIN {X -0.304,Y -654.232,Z 964.585,A 0.000,B 0.000,C 90.000,E1 321.251} C_DIS
LIN {X 0.030,Y -654.888,Z 964.578,A 0.000,B 0.000,C 90.000,E1 319.989} C_DIS
LIN {X -0.163,Y -655.611,Z 964.570,A 0.000,B 0.000,C 90.000,E1 318.528} C_DIS
LIN {X 0.011,Y -657.390,Z 964.556,A 0.000,B 0.000,C 90.000,E1 316.053} C_DIS
LIN {X -0.104,Y -658.222,Z 964.550,A 0.000,B 0.000,C 90.000,E1 315.081} C_DIS
LIN {X 0.151,Y -660.049,Z 964.538,A 0.000,B 0.000,C 90.000,E1 312.852} C_DIS
LIN {X 0.087,Y -661.137,Z 964.531,A 0.000,B 0.000,C 90.000,E1 311.634} C_DIS
LIN {X 0.022,Y -662.288,Z 964.523,A 0.000,B 0.000,C 90.000,E1 310.172} C_DIS
LIN {X -0.018,Y -663.085,Z 964.516,A 0.000,B 0.000,C 90.000,E1 308.955} C_DIS
LIN {X 0.051,Y -663.812,Z 964.510,A 0.000,B 0.000,C 90.000,E1 307.729} C_DIS
LIN {X 0.074,Y -664.184,Z 964.506,A 0.000,B 0.000,C 90.000,E1 306.996} C_DIS
LIN {X -0.234,Y -664.575,Z 964.499,A 0.000,B 0.000,C 90.000,E1 305.804} C_DIS
LIN {X 0.017,Y -664.822,Z 964.492,A 0.000,B 0.000,C 90.000,E1 304.565} C_DIS
LIN {X -0.208,Y -665.381,Z 964.483,A 0.000,B 0.000,C 90.000,E1 302.880} C_DIS
LIN {X 0.244,Y -667.121,Z 964.466,A 0.000,B 0.000,C 90.000,E1 299.922} C_DIS
LIN {X -0.104,Y -673.008,Z 964.442,A 0.000,B 0.000,C 90.000,E1 295.591} C_DIS
LIN {X 0.060,Y -675.665,Z 964.434,A 0.000,B 0.000,C 90.000,E1 294.131} C_DIS
LIN {X -0.375,Y -677.180,Z 964.429,A 0.000,B 0.000,C 90.000,E1 293.206} C_DIS
LIN {X -0.008,Y -677.753,Z 964.426,A 0.000,B 0.000,C 90.000,E1 292.695} C_DIS
LIN {X 0.101,Y -677.960,Z 964.423,A 0.000,B 0.000,C 90.000,E1 292.206} C_DIS
LIN {X 0.213,Y -677.515,Z 964.421,A 0.000,B 0.000,C 90.000,E1 291.716} C_DIS
LIN {X 0.147,Y -677.155,Z 964.419,A 0.000,B 0.000,C 90.000,E1 291.482} C_DIS
LIN {X -0.304,Y -676.165,Z 964.418,A 0.000,B 0.000,C 90.000,E1 291.280} C_DIS
LIN {X -0.284,Y -674.195,Z 964.416,A 0.000,B 0.000,C 90.000,E1 290.918} C_DIS
LIN {X -0.199,Y -673.339,Z 964.415,A 0.000,B 0.000,C 90.000,E1 290.791} C_DIS
LIN {X -0.117,Y -672.311,Z 964.415,A 0.000,B 0.000,C 90.000,E1 290.663} C_DIS
LIN {X -0.044,Y -669.296,Z 964.414,A 0.000,B 0.000,C 90.000,E1 290.429} C_DIS
LIN {X 0.016,Y -664.979,Z 964.412,A 0.000,B 0.000,C 90.000,E1 290.120} C_DIS
LIN {X -0.219,Y -658.935,Z 964.410,A 0.000,B 0.000,C 90.000,E1 289.758} C_DIS
LIN {X 0.110,Y -656.102,Z 964.409,A 0.000,B 0.000,C 90.000,E1 289.523} C_DIS
LIN {X 0.073,Y -656.080,Z 964.409,A 0.000,B 0.000,C 90.000,E1 289.523} C_DIS
LIN {X 0.177,Y -655.721,Z 964.408,A 0.000,B 0.000,C 90.000,E1 289.450} C_DIS
LIN {X 0.141,Y -655.721,Z 964.408,A 0.000,B 0.000,C 90.000,E1 289.450} C_DIS
LIN {X 0.046,Y -656.146,Z 964.406,A 0.000,B 0.000,C 90.000,E1 289.141} C_DIS
LIN {X -0.078,Y -657.056,Z 964.405,A 0.000,B 0.000,C 90.000,E1 288.906} C_DIS
LIN {X 0.011,Y -658.795,Z 964.403,A 0.000,B 0.000,C 90.000,E1 288.544} C_DIS
LIN {X -0.206,Y -664.590,Z 964.398,A 0.000,B 0.000,C 90.000,E1 287.583} C_DIS
LIN {X -0.133,Y -667.902,Z 964.394,A 0.000,B 0.000,C 90.000,E1 286.968} C_DIS
LIN {X -0.291,Y -670.202,Z 964.392,A 0.000,B 0.000,C 90.000,E1 286.496} C_DIS
LIN {X 0.211,Y -672.273,Z 964.389,A 0.000,B 0.000,C 90.000,E1 285.969} C_DIS
LIN {X 0.206,Y -674.579,Z 964.385,A 0.000,B 0.000,C 90.000,E1 285.245} C_DIS
LIN {X 0.095,Y -675.866,Z 964.382,A 0.000,B 0.000,C 90.000,E1 284.773} C_DIS
LIN {X -0.055,Y -677.361,Z 964.378,A 0.000,B 0.000,C 90.000,E1 284.064} C_DIS
LIN {X -0.233,Y -678.810,Z 964.373,A 0.000,B 0.000,C 90.000,E1 283.119} C_DIS
LIN {X 0.304,Y -679.541,Z 964.369,A 0.000,B 0.000,C 90.000,E1 282.355} C_DIS
LIN {X 0.222,Y -679.868,Z 964.366,A 0.000,B 0.000,C 90.000,E1 281.883} C_DIS
LIN {X 0.005,Y -679.949,Z 964.364,A 0.000,B 0.000,C 90.000,E1 281.422} C_DIS
LIN {X -0.118,Y -679.655,Z 964.359,A 0.000,B 0.000,C 90.000,E1 280.715} C_DIS
LIN {X -0.329,Y -679.197,Z 964.357,A 0.000,B 0.000,C 90.000,E1 280.254} C_DIS
LIN {X 0.085,Y -677.900,Z 964.353,A 0.000,B 0.000,C 90.000,E1 279.500} C_DIS
LIN {X -0.019,Y -676.728,Z 964.350,A 0.000,B 0.000,C 90.000,E1 279.029} C_DIS
LIN {X -0.240,Y -675.209,Z 964.348,A 0.000,B 0.000,C 90.000,E1 278.568} C_DIS
LIN {X 0.131,Y -672.399,Z 964.344,A 0.000,B 0.000,C 90.000,E1 277.814} C_DIS
LIN {X -0.034,Y -671.359,Z 964.342,A 0.000,B 0.000,C 90.000,E1 277.587} C_DIS
LIN {X -0.282,Y -668.297,Z 964.339,A 0.000,B 0.000,C 90.000,E1 277.004} C_DIS
LIN {X 0.019,Y -664.777,Z 964.335,A 0.000,B 0.000,C 90.000,E1 276.372} C_DIS
LIN {X 0.291,Y -660.606,Z 964.332,A 0.000,B 0.000,C 90.000,E1 275.739} C_DIS
LIN {X -0.029,Y -656.850,Z 964.329,A 0.000,B 0.000,C 90.000,E1 275.277} C_DIS
LIN {X 0.279,Y -652.679,Z 964.327,A 0.000,B 0.000,C 90.000,E1 274.759} C_DIS
LIN {X -0.250,Y -646.952,Z 964.323,A 0.000,B 0.000,C 90.000,E1 274.188} C_DIS
LIN {X 0.019,Y -642.069,Z 964.320,A 0.000,B 0.000,C 90.000,E1 273.669} C_DIS
LIN {X -0.275,Y -636.911,Z 964.318,A 0.000,B 0.000,C 90.000,E1 273.212} C_DIS
LIN {X -0.228,Y -630.120,Z 964.315,A 0.000,B 0.000,C 90.000,E1 272.636} C_DIS
LIN {X 0.014,Y -622.906,Z 964.312,A 0.000,B 0.000,C 90.000,E1 272.064} C_DIS
LIN {X -0.068,Y -616.912,Z 964.309,A 0.000,B 0.000,C 90.000,E1 271.661} C_DIS
LIN {X 0.062,Y -610.713,Z 964.307,A 0.000,B 0.000,C 90.000,E1 271.260} C_DIS
LIN {X -0.180,Y -604.077,Z 964.305,A 0.000,B 0.000,C 90.000,E1 270.917} C_DIS
LIN {X -0.068,Y -597.192,Z 964.303,A 0.000,B 0.000,C 90.000,E1 270.573} C_DIS
LIN {X -0.104,Y -590.337,Z 964.302,A 0.000,B 0.000,C 90.000,E1 270.286} C_DIS
LIN {X 0.131,Y -584.813,Z 964.300,A 0.000,B 0.000,C 90.000,E1 270.057} C_DIS
LIN {X 0.115,Y -577.420,Z 964.299,A 0.000,B 0.000,C 90.000,E1 269.828} C_DIS
LIN {X -0.218,Y -571.887,Z 964.298,A 0.000,B 0.000,C 90.000,E1 269.714} C_DIS
LIN {X 0.195,Y -565.455,Z 964.298,A 0.000,B 0.000,C 90.000,E1 269.542} C_DIS
LIN {X -0.264,Y -557.606,Z 964.297,A 0.000,B 0.000,C 90.000,E1 269.484} C_DIS
LIN {X 0.046,Y -547.326,Z 964.297,A 0.000,B 0.000,C 90.000,E1 269.427} C_DIS
LIN {X -0.114,Y -544.181,Z 964.296,A 0.000,B 0.000,C 90.000,E1 269.312} C_DIS
LIN {X -0.266,Y -543.666,Z 964.296,A 0.000,B 0.000,C 90.000,E1 269.312} C_DIS
LIN {X 0.227,Y -543.559,Z 964.296,A 0.000,B 0.000,C 90.000,E1 269.255} C_DIS
LIN {X -0.018,Y -542.849,Z 964.295,A 0.000,B 0.000,C 90.000,E1 269.026} C_DIS
LIN {X -0.117,Y -542.623,Z 964.293,A 0.000,B 0.000,C 90.000,E1 268.682} C_DIS
LIN {X 0.192,Y -540.415,Z 964.277,A 0.000,B 0.000,C 90.000,E1 265.812} C_DIS
LIN {X -0.197,Y -539.431,Z 964.269,A 0.000,B 0.000,C 90.000,E1 264.432} C_DIS
LIN {X -0.073,Y -538.620,Z 964.263,A 0.000,B 0.000,C 90.000,E1 263.280} C_DIS
LIN {X 0.091,Y -537.412,Z 964.255,A 0.000,B 0.000,C 90.000,E1 261.837} C_DIS
LIN {X 0.189,Y -536.527,Z 964.250,A 0.000,B 0.000,C 90.000,E1 260.971} C_DIS
LIN {X -0.107,Y -535.333,Z 964.244,A 0.000,B 0.000,C 90.000,E1 259.859} C_DIS
LIN {X 0.063,Y -533.585,Z 964.236,A 0.000,B 0.000,C 90.000,E1 258.409} C_DIS
LIN {X -0.152,Y -532.241,Z 964.229,A 0.000,B 0.000,C 90.000,E1 257.285} C_DIS
LIN {X -0.230,Y -529.478,Z 964.217,A 0.000,B 0.000,C 90.000,E1 254.991} C_DIS
LIN {X 0.178,Y -527.947,Z 964.208,A 0.000,B 0.000,C 90.000,E1 253.504} C_DIS
LIN {X 0.207,Y -526.325,Z 964.201,A 0.000,B 0.000,C 90.000,E1 252.054} C_DIS
LIN {X -0.294,Y -524.089,Z 964.191,A 0.000,B 0.000,C 90.000,E1 250.369} C_DIS
LIN {X -0.160,Y -522.190,Z 964.183,A 0.000,B 0.000,C 90.000,E1 248.901} C_DIS
LIN {X 0.132,Y -520.382,Z 964.175,A 0.000,B 0.000,C 90.000,E1 247.411} C_DIS
LIN {X 0.056,Y -517.786,Z 964.165,A 0.000,B 0.000,C 90.000,E1 245.665} C_DIS
LIN {X 0.120,Y -515.972,Z 964.158,A 0.000,B 0.000,C 90.000,E1 244.485} C_DIS
LIN {X -0.090,Y -513.237,Z 964.149,A 0.000,B 0.000,C 90.000,E1 242.743} C_DIS
LIN {X 0.000,Y -510.844,Z 964.140,A 0.000,B 0.000,C 90.000,E1 241.257} C_DIS
LIN {X -0.045,Y -508.852,Z 964.134,A 0.000,B 0.000,C 90.000,E1 240.078} C_DIS
LIN {X 0.135,Y -506.611,Z 964.127,A 0.000,B 0.000,C 90.000,E1 238.869} C_DIS
LIN {X -0.142,Y -504.219,Z 964.121,A 0.000,B 0.000,C 90.000,E1 237.709} C_DIS
LIN {X -0.030,Y -501.667,Z 964.114,A 0.000,B 0.000,C 90.000,E1 236.501} C_DIS
LIN {X 0.056,Y -497.515,Z 964.104,A 0.000,B 0.000,C 90.000,E1 234.689} C_DIS
LIN {X -0.057,Y -493.513,Z 964.094,A 0.000,B 0.000,C 90.000,E1 232.889} C_DIS
LIN {X 0.124,Y -489.332,Z 964.084,A 0.000,B 0.000,C 90.000,E1 231.045} C_DIS
LIN {X 0.019,Y -483.653,Z 964.070,A 0.000,B 0.000,C 90.000,E1 228.609} C_DIS
LIN {X 0.072,Y -478.079,Z 964.056,A 0.000,B 0.000,C 90.000,E1 226.134} C_DIS
LIN {X -0.039,Y -474.679,Z 964.048,A 0.000,B 0.000,C 90.000,E1 224.595} C_DIS
LIN {X 0.217,Y -470.540,Z 964.037,A 0.000,B 0.000,C 90.000,E1 222.690} C_DIS
LIN {X 0.049,Y -466.357,Z 964.027,A 0.000,B 0.000,C 90.000,E1 220.825} C_DIS
LIN {X 0.033,Y -463.641,Z 964.020,A 0.000,B 0.000,C 90.000,E1 219.564} C_DIS
LIN {X -0.045,Y -457.989,Z 964.006,A 0.000,B 0.000,C 90.000,E1 217.030} C_DIS
LIN {X -0.009,Y -453.662,Z 963.995,A 0.000,B 0.000,C 90.000,E1 215.105} C_DIS
LIN {X 0.113,Y -448.718,Z 963.983,A 0.000,B 0.000,C 90.000,E1 212.832} C_DIS
LIN {X -0.209,Y -444.568,Z 963.972,A 0.000,B 0.000,C 90.000,E1 210.924} C_DIS
LIN {X -0.053,Y -439.559,Z 963.959,A 0.000,B 0.000,C 90.000,E1 208.615} C_DIS
LIN {X 0.116,Y -435.255,Z 963.948,A 0.000,B 0.000,C 90.000,E1 206.616} C_DIS
LIN {X 0.174,Y -432.329,Z 963.941,A 0.000,B 0.000,C 90.000,E1 205.283} C_DIS
LIN {X -0.008,Y -428.453,Z 963.931,A 0.000,B 0.000,C 90.000,E1 203.643} C_DIS
LIN {X 0.067,Y -421.737,Z 963.915,A 0.000,B 0.000,C 90.000,E1 200.610} C_DIS
LIN {X 0.144,Y -418.172,Z 963.905,A 0.000,B 0.000,C 90.000,E1 198.906} C_DIS
LIN {X 0.165,Y -414.077,Z 963.894,A 0.000,B 0.000,C 90.000,E1 196.858} C_DIS
LIN {X 0.213,Y -411.454,Z 963.886,A 0.000,B 0.000,C 90.000,E1 195.481} C_DIS
LIN {X 0.123,Y -408.063,Z 963.877,A 0.000,B 0.000,C 90.000,E1 193.772} C_DIS
LIN {X -0.030,Y -404.676,Z 963.867,A 0.000,B 0.000,C 90.000,E1 192.063} C_DIS
LIN {X 0.050,Y -400.715,Z 963.855,A 0.000,B 0.000,C 90.000,E1 189.962} C_DIS
LIN {X -0.017,Y -397.359,Z 963.846,A 0.000,B 0.000,C 90.000,E1 188.219} C_DIS
LIN {X 0.119,Y -390.049,Z 963.822,A 0.000,B 0.000,C 90.000,E1 183.955} C_DIS
LIN {X -0.058,Y -389.178,Z 963.818,A 0.000,B 0.000,C 90.000,E1 183.269} C_DIS
LIN {X 0.169,Y -388.642,Z 963.814,A 0.000,B 0.000,C 90.000,E1 182.522} C_DIS
LIN {X -0.046,Y -388.484,Z 963.809,A 0.000,B 0.000,C 90.000,E1 181.661} C_DIS
LIN {X 0.044,Y -388.875,Z 963.807,A 0.000,B 0.000,C 90.000,E1 181.260} C_DIS
LIN {X -0.093,Y -389.218,Z 963.804,A 0.000,B 0.000,C 90.000,E1 180.745} C_DIS
LIN {X -0.139,Y -389.472,Z 963.803,A 0.000,B 0.000,C 90.000,E1 180.573} C_DIS
LIN {X 0.037,Y -391.101,Z 963.800,A 0.000,B 0.000,C 90.000,E1 179.943} C_DIS
LIN {X -0.096,Y -393.495,Z 963.796,A 0.000,B 0.000,C 90.000,E1 179.370} C_DIS
LIN {X -0.134,Y -394.386,Z 963.795,A 0.000,B 0.000,C 90.000,E1 179.198} C_DIS
LIN {X 0.154,Y -397.819,Z 963.793,A 0.000,B 0.000,C 90.000,E1 178.625} C_DIS
LIN {X 0.063,Y -400.155,Z 963.791,A 0.000,B 0.000,C 90.000,E1 178.339} C_DIS
LIN {X -0.118,Y -403.910,Z 963.789,A 0.000,B 0.000,C 90.000,E1 177.936} C_DIS
LIN {X 0.007,Y -421.972,Z 963.779,A 0.000,B 0.000,C 90.000,E1 176.274} C_DIS
LIN {X 0.142,Y -432.680,Z 963.774,A 0.000,B 0.000,C 90.000,E1 175.298} C_DIS
LIN {X -0.030,Y -438.698,Z 963.771,A 0.000,B 0.000,C 90.000,E1 174.780} C_DIS
LIN {X 0.149,Y -447.556,Z 963.766,A 0.000,B 0.000,C 90.000,E1 173.913} C_DIS
LIN {X -0.181,Y -453.296,Z 963.763,A 0.000,B 0.000,C 90.000,E1 173.394} C_DIS
LIN {X 0.219,Y -458.987,Z 963.760,A 0.000,B 0.000,C 90.000,E1 172.761} C_DIS
LIN {X 0.161,Y -468.549,Z 963.754,A 0.000,B 0.000,C 90.000,E1 171.724} C_DIS
LIN {X -0.065,Y -476.637,Z 963.749,A 0.000,B 0.000,C 90.000,E1 170.849} C_DIS
LIN {X 0.129,Y -485.387,Z 963.743,A 0.000,B 0.000,C 90.000,E1 169.746} C_DIS
LIN {X -0.124,Y -490.241,Z 963.740,A 0.000,B 0.000,C 90.000,E1 169.162} C_DIS
LIN {X 0.046,Y -497.291,Z 963.735,A 0.000,B 0.000,C 90.000,E1 168.229} C_DIS
LIN {X 0.141,Y -502.725,Z 963.731,A 0.000,B 0.000,C 90.000,E1 167.465} C_DIS
LIN {X 0.239,Y -510.097,Z 963.725,A 0.000,B 0.000,C 90.000,E1 166.408} C_DIS
LIN {X -0.229,Y -517.877,Z 963.718,A 0.000,B 0.000,C 90.000,E1 165.283} C_DIS
LIN {X 0.195,Y -524.305,Z 963.712,A 0.000,B 0.000,C 90.000,E1 164.212} C_DIS
LIN {X -0.136,Y -529.768,Z 963.708,A 0.000,B 0.000,C 90.000,E1 163.378} C_DIS
LIN {X 0.136,Y -537.618,Z 963.700,A 0.000,B 0.000,C 90.000,E1 162.054} C_DIS
LIN {X -0.207,Y -543.608,Z 963.695,A 0.000,B 0.000,C 90.000,E1 161.094} C_DIS
LIN {X 0.036,Y -552.774,Z 963.686,A 0.000,B 0.000,C 90.000,E1 159.518} C_DIS
LIN {X -0.058,Y -559.242,Z 963.680,A 0.000,B 0.000,C 90.000,E1 158.411} C_DIS
LIN {X 0.252,Y -564.428,Z 963.675,A 0.000,B 0.000,C 90.000,E1 157.411} C_DIS
LIN {X -0.020,Y -568.818,Z 963.670,A 0.000,B 0.000,C 90.000,E1 156.613} C_DIS
LIN {X 0.091,Y -576.213,Z 963.662,A 0.000,B 0.000,C 90.000,E1 155.101} C_DIS
LIN {X -0.211,Y -578.733,Z 963.659,A 0.000,B 0.000,C 90.000,E1 154.588} C_DIS
LIN {X 0.139,Y -584.528,Z 963.651,A 0.000,B 0.000,C 90.000,E1 153.204} C_DIS
LIN {X 0.037,Y -587.783,Z 963.647,A 0.000,B 0.000,C 90.000,E1 152.410} C_DIS
LIN {X -0.304,Y -590.648,Z 963.642,A 0.000,B 0.000,C 90.000,E1 151.641} C_DIS
LIN {X 0.081,Y -594.310,Z 963.636,A 0.000,B 0.000,C 90.000,E1 150.539} C_DIS
LIN {X 0.210,Y -598.752,Z 963.629,A 0.000,B 0.000,C 90.000,E1 149.203} C_DIS
LIN {X -0.092,Y -603.102,Z 963.622,A 0.000,B 0.000,C 90.000,E1 147.916} C_DIS
LIN {X 0.002,Y -605.614,Z 963.617,A 0.000,B 0.000,C 90.000,E1 147.120} C_DIS
LIN {X -0.057,Y -608.090,Z 963.613,A 0.000,B 0.000,C 90.000,E1 146.342} C_DIS
LIN {X -0.146,Y -611.510,Z 963.607,A 0.000,B 0.000,C 90.000,E1 145.308} C_DIS
LIN {X 0.101,Y -615.734,Z 963.600,A 0.000,B 0.000,C 90.000,E1 143.989} C_DIS
LIN {X 0.057,Y -621.453,Z 963.590,A 0.000,B 0.000,C 90.000,E1 142.190} C_DIS
LIN {X -0.143,Y -625.542,Z 963.583,A 0.000,B 0.000,C 90.000,E1 140.928} C_DIS
LIN {X 0.308,Y -631.997,Z 963.572,A 0.000,B 0.000,C 90.000,E1 138.852} C_DIS
LIN {X -0.035,Y -638.722,Z 963.560,A 0.000,B 0.000,C 90.000,E1 136.863} C_DIS
LIN {X 0.210,Y -645.545,Z 963.549,A 0.000,B 0.000,C 90.000,E1 134.838} C_DIS
LIN {X 0.148,Y -653.426,Z 963.537,A 0.000,B 0.000,C 90.000,E1 132.609} C_DIS
LIN {X -0.077,Y -661.601,Z 963.525,A 0.000,B 0.000,C 90.000,E1 130.415} C_DIS
LIN {X -0.089,Y -665.310,Z 963.519,A 0.000,B 0.000,C 90.000,E1 129.439} C_DIS
LIN {X -0.043,Y -668.029,Z 963.515,A 0.000,B 0.000,C 90.000,E1 128.705} C_DIS
LIN {X -0.401,Y -672.363,Z 963.508,A 0.000,B 0.000,C 90.000,E1 127.523} C_DIS
LIN {X -0.164,Y -676.515,Z 963.502,A 0.000,B 0.000,C 90.000,E1 126.297} C_DIS
LIN {X -0.260,Y -680.353,Z 963.495,A 0.000,B 0.000,C 90.000,E1 125.105} C_DIS
LIN {X 0.086,Y -683.238,Z 963.490,A 0.000,B 0.000,C 90.000,E1 124.119} C_DIS
LIN {X 0.086,Y -685.858,Z 963.484,A 0.000,B 0.000,C 90.000,E1 123.166} C_DIS
LIN {X -0.029,Y -689.643,Z 963.476,A 0.000,B 0.000,C 90.000,E1 121.750} C_DIS
LIN {X -0.309,Y -692.419,Z 963.470,A 0.000,B 0.000,C 90.000,E1 120.590} C_DIS
LIN {X -0.194,Y -693.886,Z 963.466,A 0.000,B 0.000,C 90.000,E1 119.873} C_DIS
LIN {X -0.059,Y -695.217,Z 963.462,A 0.000,B 0.000,C 90.000,E1 119.155} C_DIS
LIN {X -0.009,Y -696.699,Z 963.455,A 0.000,B 0.000,C 90.000,E1 117.975} C_DIS
LIN {X 0.152,Y -697.495,Z 963.452,A 0.000,B 0.000,C 90.000,E1 117.257} C_DIS
LIN {X -0.093,Y -698.414,Z 963.445,A 0.000,B 0.000,C 90.000,E1 116.104} C_DIS
LIN {X 0.304,Y -698.939,Z 963.439,A 0.000,B 0.000,C 90.000,E1 114.899} C_DIS
LIN {X 0.175,Y -698.989,Z 963.435,A 0.000,B 0.000,C 90.000,E1 114.207} C_DIS
LIN {X -0.217,Y -698.641,Z 963.432,A 0.000,B 0.000,C 90.000,E1 113.770} C_DIS
LIN {X 0.307,Y -697.526,Z 963.429,A 0.000,B 0.000,C 90.000,E1 113.259} C_DIS
LIN {X -0.351,Y -696.855,Z 963.428,A 0.000,B 0.000,C 90.000,E1 113.078} C_DIS
LIN {X -0.223,Y -696.234,Z 963.427,A 0.000,B 0.000,C 90.000,E1 112.950} C_DIS
LIN {X 0.010,Y -692.605,Z 963.425,A 0.000,B 0.000,C 90.000,E1 112.461} C_DIS
LIN {X 0.131,Y -691.533,Z 963.424,A 0.000,B 0.000,C 90.000,E1 112.333} C_DIS
LIN {X 0.248,Y -689.905,Z 963.424,A 0.000,B 0.000,C 90.000,E1 112.206} C_DIS
LIN {X 0.092,Y -685.740,Z 963.422,A 0.000,B 0.000,C 90.000,E1 112.025} C_DIS
LIN {X -0.196,Y -680.147,Z 963.421,A 0.000,B 0.000,C 90.000,E1 111.844} C_DIS
LIN {X -0.097,Y -675.557,Z 963.421,A 0.000,B 0.000,C 90.000,E1 111.716} C_DIS
LIN {X 0.160,Y -670.699,Z 963.420,A 0.000,B 0.000,C 90.000,E1 111.663} C_DIS
LIN {X 0.041,Y -668.146,Z 963.420,A 0.000,B 0.000,C 90.000,E1 111.663} C_DIS
LIN {X -0.008,Y -628.532,Z 963.420,A 0.000,B 0.000,C 90.000,E1 111.663} C_DIS
LIN {X 0.273,Y -622.220,Z 963.420,A 0.000,B 0.000,C 90.000,E1 111.535} C_DIS
LIN {X 0.276,Y -616.971,Z 963.419,A 0.000,B 0.000,C 90.000,E1 111.408} C_DIS
LIN {X -0.054,Y -608.349,Z 963.418,A 0.000,B 0.000,C 90.000,E1 111.153} C_DIS
LIN {X 0.113,Y -604.522,Z 963.417,A 0.000,B 0.000,C 90.000,E1 110.972} C_DIS
LIN {X 0.035,Y -598.476,Z 963.415,A 0.000,B 0.000,C 90.000,E1 110.663} C_DIS
LIN {X 0.086,Y -591.291,Z 963.412,A 0.000,B 0.000,C 90.000,E1 110.194} C_DIS
LIN {X -0.087,Y -575.509,Z 963.406,A 0.000,B 0.000,C 90.000,E1 109.033} C_DIS
LIN {X -0.083,Y -567.267,Z 963.403,A 0.000,B 0.000,C 90.000,E1 108.544} C_DIS
LIN {X 0.257,Y -553.172,Z 963.399,A 0.000,B 0.000,C 90.000,E1 107.819} C_DIS
LIN {X -0.199,Y -550.746,Z 963.398,A 0.000,B 0.000,C 90.000,E1 107.638} C_DIS
LIN {X -0.238,Y -550.721,Z 963.398,A 0.000,B 0.000,C 90.000,E1 107.638} C_DIS
LIN {X -0.001,Y -550.342,Z 963.397,A 0.000,B 0.000,C 90.000,E1 107.457} C_DIS
LIN {X 0.097,Y -550.196,Z 963.395,A 0.000,B 0.000,C 90.000,E1 107.166} C_DIS
LIN {X -0.071,Y -550.300,Z 963.392,A 0.000,B 0.000,C 90.000,E1 106.622} C_DIS
LIN {X 0.219,Y -550.852,Z 963.385,A 0.000,B 0.000,C 90.000,E1 105.190} C_DIS
LIN {X 0.187,Y -552.016,Z 963.372,A 0.000,B 0.000,C 90.000,E1 102.952} C_DIS
LIN {X 0.034,Y -554.809,Z 963.353,A 0.000,B 0.000,C 90.000,E1 99.613} C_DIS
LIN {X 0.215,Y -556.666,Z 963.343,A 0.000,B 0.000,C 90.000,E1 97.644} C_DIS
LIN {X 0.043,Y -557.617,Z 963.336,A 0.000,B 0.000,C 90.000,E1 96.549} C_DIS
LIN {X 0.013,Y -558.655,Z 963.329,A 0.000,B 0.000,C 90.000,E1 95.163} C_DIS
LIN {X -0.262,Y -559.193,Z 963.324,A 0.000,B 0.000,C 90.000,E1 94.359} C_DIS
LIN {X -0.237,Y -560.148,Z 963.315,A 0.000,B 0.000,C 90.000,E1 92.694} C_DIS
LIN {X -0.223,Y -560.992,Z 963.306,A 0.000,B 0.000,C 90.000,E1 91.031} C_DIS
LIN {X 0.164,Y -561.468,Z 963.299,A 0.000,B 0.000,C 90.000,E1 89.885} C_DIS
LIN {X 0.093,Y -561.885,Z 963.292,A 0.000,B 0.000,C 90.000,E1 88.511} C_DIS
LIN {X 0.041,Y -562.188,Z 963.284,A 0.000,B 0.000,C 90.000,E1 87.135} C_DIS
LIN {X -0.105,Y -562.400,Z 963.278,A 0.000,B 0.000,C 90.000,E1 86.045} C_DIS
LIN {X 0.028,Y -562.622,Z 963.269,A 0.000,B 0.000,C 90.000,E1 84.375} C_DIS
LIN {X -0.062,Y -562.787,Z 963.263,A 0.000,B 0.000,C 90.000,E1 83.280} C_DIS
LIN {X 0.230,Y -563.173,Z 963.252,A 0.000,B 0.000,C 90.000,E1 81.319} C_DIS
LIN {X -0.087,Y -564.086,Z 963.238,A 0.000,B 0.000,C 90.000,E1 78.870} C_DIS
LIN {X -0.033,Y -565.058,Z 963.227,A 0.000,B 0.000,C 90.000,E1 76.937} C_DIS
LIN {X -0.163,Y -565.941,Z 963.220,A 0.000,B 0.000,C 90.000,E1 75.574} C_DIS
LIN {X 0.212,Y -567.251,Z 963.209,A 0.000,B 0.000,C 90.000,E1 73.614} C_DIS
LIN {X -0.102,Y -568.326,Z 963.200,A 0.000,B 0.000,C 90.000,E1 72.000} C_DIS
LIN {X -0.229,Y -569.254,Z 963.191,A 0.000,B 0.000,C 90.000,E1 70.369} C_DIS
LIN {X -0.149,Y -569.996,Z 963.182,A 0.000,B 0.000,C 90.000,E1 68.720} C_DIS
LIN {X -0.157,Y -570.329,Z 963.177,A 0.000,B 0.000,C 90.000,E1 67.901} C_DIS
LIN {X 0.159,Y -570.875,Z 963.168,A 0.000,B 0.000,C 90.000,E1 66.230} C_DIS
LIN {X 0.355,Y -571.222,Z 963.161,A 0.000,B 0.000,C 90.000,E1 64.845} C_DIS
LIN {X -0.128,Y -571.580,Z 963.151,A 0.000,B 0.000,C 90.000,E1 63.256} C_DIS
LIN {X 0.152,Y -571.800,Z 963.142,A 0.000,B 0.000,C 90.000,E1 61.591} C_DIS
LIN {X -0.128,Y -571.890,Z 963.135,A 0.000,B 0.000,C 90.000,E1 60.255} C_DIS
LIN {X -0.078,Y -572.093,Z 963.126,A 0.000,B 0.000,C 90.000,E1 58.614} C_DIS
LIN {X -0.046,Y -572.170,Z 963.118,A 0.000,B 0.000,C 90.000,E1 57.248} C_DIS
LIN {X -0.011,Y -571.966,Z 963.110,A 0.000,B 0.000,C 90.000,E1 55.881} C_DIS
LIN {X -0.126,Y -571.669,Z 963.103,A 0.000,B 0.000,C 90.000,E1 54.529} C_DIS
LIN {X -0.186,Y -571.542,Z 963.100,A 0.000,B 0.000,C 90.000,E1 53.989} C_DIS
LIN {X -0.099,Y -570.971,Z 963.094,A 0.000,B 0.000,C 90.000,E1 52.889} C_DIS
LIN {X -0.044,Y -570.449,Z 963.089,A 0.000,B 0.000,C 90.000,E1 52.065} C_DIS
LIN {X -0.100,Y -569.772,Z 963.085,A 0.000,B 0.000,C 90.000,E1 51.251} C_DIS
LIN {X -0.351,Y -568.487,Z 963.077,A 0.000,B 0.000,C 90.000,E1 49.908} C_DIS
LIN {X -0.055,Y -567.494,Z 963.073,A 0.000,B 0.000,C 90.000,E1 49.057} C_DIS
LIN {X -0.142,Y -566.328,Z 963.068,A 0.000,B 0.000,C 90.000,E1 48.243} C_DIS
LIN {X 0.131,Y -564.965,Z 963.063,A 0.000,B 0.000,C 90.000,E1 47.391} C_DIS
LIN {X -0.254,Y -562.295,Z 963.056,A 0.000,B 0.000,C 90.000,E1 46.053} C_DIS
LIN {X 0.034,Y -559.683,Z 963.050,A 0.000,B 0.000,C 90.000,E1 44.919} C_DIS
LIN {X 0.165,Y -558.288,Z 963.047,A 0.000,B 0.000,C 90.000,E1 44.352} C_DIS
LIN {X 0.007,Y -554.909,Z 963.040,A 0.000,B 0.000,C 90.000,E1 43.257} C_DIS
LIN {X 0.100,Y -553.037,Z 963.037,A 0.000,B 0.000,C 90.000,E1 42.690} C_DIS
LIN {X 0.227,Y -549.937,Z 963.033,A 0.000,B 0.000,C 90.000,E1 41.838} C_DIS
LIN {X -0.041,Y -546.600,Z 963.028,A 0.000,B 0.000,C 90.000,E1 41.024} C_DIS
LIN {X -0.180,Y -543.380,Z 963.024,A 0.000,B 0.000,C 90.000,E1 40.334} C_DIS
LIN {X -0.352,Y -539.884,Z 963.020,A 0.000,B 0.000,C 90.000,E1 39.644} C_DIS
LIN {X -0.134,Y -534.645,Z 963.015,A 0.000,B 0.000,C 90.000,E1 38.624} C_DIS
LIN {X 0.185,Y -529.692,Z 963.010,A 0.000,B 0.000,C 90.000,E1 37.729} C_DIS
LIN {X -0.051,Y -523.660,Z 963.004,A 0.000,B 0.000,C 90.000,E1 36.744} C_DIS
LIN {X 0.001,Y -519.080,Z 963.000,A 0.000,B 0.000,C 90.000,E1 36.011} C_DIS
LIN {X 0.241,Y -513.398,Z 962.995,A 0.000,B 0.000,C 90.000,E1 35.105} C_DIS
LIN {X -0.102,Y -508.179,Z 962.991,A 0.000,B 0.000,C 90.000,E1 34.405} C_DIS
LIN {X -0.071,Y -502.558,Z 962.987,A 0.000,B 0.000,C 90.000,E1 33.658} C_DIS
LIN {X -0.106,Y -498.943,Z 962.984,A 0.000,B 0.000,C 90.000,E1 33.214} C_DIS
LIN {X -0.020,Y -495.223,Z 962.982,A 0.000,B 0.000,C 90.000,E1 32.752} C_DIS
LIN {X -0.093,Y -487.104,Z 962.977,A 0.000,B 0.000,C 90.000,E1 31.878} C_DIS
LIN {X 0.268,Y -481.516,Z 962.974,A 0.000,B 0.000,C 90.000,E1 31.258} C_DIS
LIN {X -0.150,Y -471.374,Z 962.969,A 0.000,B 0.000,C 90.000,E1 30.335} C_DIS
LIN {X 0.109,Y -463.971,Z 962.965,A 0.000,B 0.000,C 90.000,E1 29.617} C_DIS
LIN {X 0.061,Y -453.510,Z 962.959,A 0.000,B 0.000,C 90.000,E1 28.693} C_DIS
LIN {X 0.171,Y -441.281,Z 962.954,A 0.000,B 0.000,C 90.000,E1 27.641} C_DIS
LIN {X 0.014,Y -418.713,Z 962.943,A 0.000,B 0.000,C 90.000,E1 25.668} C_DIS
LIN {X 0.156,Y -404.042,Z 962.935,A 0.000,B 0.000,C 90.000,E1 24.207} C_DIS
LIN {X -0.067,Y -397.066,Z 962.930,A 0.000,B 0.000,C 90.000,E1 23.462} C_DIS
LIN {X 0.011,Y -394.785,Z 962.929,A 0.000,B 0.000,C 90.000,E1 23.153} C_DIS
LIN {X -0.048,Y -393.739,Z 962.928,A 0.000,B 0.000,C 90.000,E1 23.003} C_DIS
LIN {X 0.148,Y -391.224,Z 962.925,A 0.000,B 0.000,C 90.000,E1 22.461} C_DIS
LIN {X -0.229,Y -390.227,Z 962.923,A 0.000,B 0.000,C 90.000,E1 22.153} C_DIS
LIN {X -0.041,Y -389.842,Z 962.921,A 0.000,B 0.000,C 90.000,E1 21.770} C_DIS
LIN {X -0.004,Y -389.586,Z 962.919,A 0.000,B 0.000,C 90.000,E1 21.408} C_DIS
LIN {X -0.118,Y -389.891,Z 962.913,A 0.000,B 0.000,C 90.000,E1 20.355} C_DIS
LIN {X -0.108,Y -393.618,Z 962.891,A 0.000,B 0.000,C 90.000,E1 16.441} C_DIS
LIN {X 0.076,Y -396.659,Z 962.878,A 0.000,B 0.000,C 90.000,E1 13.939} C_DIS
LIN {X 0.021,Y -401.706,Z 962.858,A 0.000,B 0.000,C 90.000,E1 10.433} C_DIS
LIN {X 0.034,Y -407.139,Z 962.841,A 0.000,B 0.000,C 90.000,E1 7.296} C_DIS
LIN {X 0.017,Y -410.436,Z 962.831,A 0.000,B 0.000,C 90.000,E1 5.568} C_DIS
LIN {X 0.106,Y -416.151,Z 962.816,A 0.000,B 0.000,C 90.000,E1 2.808} C_DIS
LIN {X -0.202,Y -419.979,Z 962.806,A 0.000,B 0.000,C 90.000,E1 1.146} C_DIS
LIN {X -0.103,Y -422.439,Z 962.801,A 0.000,B 0.000,C 90.000,E1 0.115} C_DIS
LIN {X 0.161,Y -423.382,Z 962.799,A 0.000,B 0.000,C 90.000,E1 359.771} C_DIS
LIN {X -0.052,Y -425.251,Z 962.796,A 0.000,B 0.000,C 90.000,E1 359.312} C_DIS
LIN {X 0.036,Y -429.597,Z 962.792,A 0.000,B 0.000,C 90.000,E1 358.568} C_DIS
LIN {X -0.169,Y -434.260,Z 962.790,A 0.000,B 0.000,C 90.000,E1 358.165} C_DIS
LIN {X -0.068,Y -438.459,Z 962.788,A 0.000,B 0.000,C 90.000,E1 357.879} C_DIS
LIN {X 0.217,Y -454.972,Z 962.783,A 0.000,B 0.000,C 90.000,E1 356.963} C_DIS
LIN {X -0.092,Y -471.897,Z 962.778,A 0.000,B 0.000,C 90.000,E1 356.102} C_DIS
LIN {X -0.156,Y -483.402,Z 962.775,A 0.000,B 0.000,C 90.000,E1 355.469} C_DIS
LIN {X 0.181,Y -495.167,Z 962.771,A 0.000,B 0.000,C 90.000,E1 354.780} C_DIS
LIN {X -0.174,Y -504.828,Z 962.768,A 0.000,B 0.000,C 90.000,E1 354.261} C_DIS
LIN {X -0.199,Y -515.788,Z 962.764,A 0.000,B 0.000,C 90.000,E1 353.571} C_DIS
LIN {X -0.106,Y -523.547,Z 962.761,A 0.000,B 0.000,C 90.000,E1 353.053} C_DIS
LIN {X -0.215,Y -532.500,Z 962.758,A 0.000,B 0.000,C 90.000,E1 352.413} C_DIS
LIN {X 0.183,Y -539.638,Z 962.755,A 0.000,B 0.000,C 90.000,E1 351.781} C_DIS
LIN {X -0.098,Y -545.237,Z 962.752,A 0.000,B 0.000,C 90.000,E1 351.319} C_DIS
LIN {X -0.085,Y -551.817,Z 962.748,A 0.000,B 0.000,C 90.000,E1 350.679} C_DIS
LIN {X -0.123,Y -556.968,Z 962.745,A 0.000,B 0.000,C 90.000,E1 350.151} C_DIS
LIN {X -0.020,Y -562.704,Z 962.741,A 0.000,B 0.000,C 90.000,E1 349.454} C_DIS
LIN {X 0.300,Y -567.065,Z 962.738,A 0.000,B 0.000,C 90.000,E1 348.870} C_DIS
LIN {X -0.148,Y -571.972,Z 962.735,A 0.000,B 0.000,C 90.000,E1 348.229} C_DIS
LIN {X -0.116,Y -577.426,Z 962.730,A 0.000,B 0.000,C 90.000,E1 347.409} C_DIS
LIN {X 0.209,Y -581.560,Z 962.726,A 0.000,B 0.000,C 90.000,E1 346.700} C_DIS
LIN {X 0.007,Y -585.544,Z 962.723,A 0.000,B 0.000,C 90.000,E1 346.047} C_DIS
LIN {X -0.215,Y -592.092,Z 962.716,A 0.000,B 0.000,C 90.000,E1 344.866} C_DIS
LIN {X -0.119,Y -597.470,Z 962.710,A 0.000,B 0.000,C 90.000,E1 343.795} C_DIS
LIN {X 0.100,Y -601.902,Z 962.705,A 0.000,B 0.000,C 90.000,E1 342.851} C_DIS
LIN {X -0.077,Y -606.626,Z 962.699,A 0.000,B 0.000,C 90.000,E1 341.819} C_DIS
LIN {X -0.187,Y -611.084,Z 962.693,A 0.000,B 0.000,C 90.000,E1 340.786} C_DIS
LIN {X -0.236,Y -615.291,Z 962.687,A 0.000,B 0.000,C 90.000,E1 339.752} C_DIS
LIN {X -0.235,Y -619.246,Z 962.682,A 0.000,B 0.000,C 90.000,E1 338.720} C_DIS
LIN {X 0.055,Y -622.031,Z 962.677,A 0.000,B 0.000,C 90.000,E1 337.922} C_DIS
LIN {X -0.204,Y -625.462,Z 962.672,A 0.000,B 0.000,C 90.000,E1 336.922} C_DIS
LIN {X 0.158,Y -628.755,Z 962.666,A 0.000,B 0.000,C 90.000,E1 335.869} C_DIS
LIN {X 0.253,Y -631.856,Z 962.660,A 0.000,B 0.000,C 90.000,E1 334.845} C_DIS
LIN {X 0.118,Y -634.705,Z 962.655,A 0.000,B 0.000,C 90.000,E1 333.845} C_DIS
LIN {X -0.272,Y -637.296,Z 962.649,A 0.000,B 0.000,C 90.000,E1 332.871} C_DIS
LIN {X -0.061,Y -639.712,Z 962.644,A 0.000,B 0.000,C 90.000,E1 331.847} C_DIS
LIN {X -0.011,Y -642.529,Z 962.637,A 0.000,B 0.000,C 90.000,E1 330.589} C_DIS
LIN {X 0.023,Y -644.614,Z 962.631,A 0.000,B 0.000,C 90.000,E1 329.587} C_DIS
LIN {X -0.320,Y -646.030,Z 962.627,A 0.000,B 0.000,C 90.000,E1 328.869} C_DIS
LIN {X 0.175,Y -648.111,Z 962.620,A 0.000,B 0.000,C 90.000,E1 327.582} C_DIS
LIN {X -0.269,Y -649.566,Z 962.615,A 0.000,B 0.000,C 90.000,E1 326.628} C_DIS
LIN {X -0.262,Y -651.070,Z 962.608,A 0.000,B 0.000,C 90.000,E1 325.388} C_DIS
LIN {X -0.304,Y -652.150,Z 962.602,A 0.000,B 0.000,C 90.000,E1 324.402} C_DIS
LIN {X -0.334,Y -653.064,Z 962.597,A 0.000,B 0.000,C 90.000,E1 323.417} C_DIS
LIN {X 0.093,Y -653.962,Z 962.590,A 0.000,B 0.000,C 90.000,E1 322.145} C_DIS
LIN {X -0.090,Y -654.756,Z 962.583,A 0.000,B 0.000,C 90.000,E1 320.928} C_DIS
LIN {X 0.307,Y -655.337,Z 962.577,A 0.000,B 0.000,C 90.000,E1 319.908} C_DIS
LIN {X 0.163,Y -655.931,Z 962.571,A 0.000,B 0.000,C 90.000,E1 318.690} C_DIS
LIN {X 0.316,Y -657.860,Z 962.556,A 0.000,B 0.000,C 90.000,E1 315.972} C_DIS
LIN {X 0.183,Y -658.863,Z 962.549,A 0.000,B 0.000,C 90.000,E1 314.757} C_DIS
LIN {X 0.009,Y -660.771,Z 962.537,A 0.000,B 0.000,C 90.000,E1 312.567} C_DIS
LIN {X -0.097,Y -661.855,Z 962.530,A 0.000,B 0.000,C 90.000,E1 311.353} C_DIS
LIN {X 0.364,Y -662.803,Z 962.523,A 0.000,B 0.000,C 90.000,E1 310.092} C_DIS
LIN {X -0.086,Y -663.613,Z 962.516,A 0.000,B 0.000,C 90.000,E1 308.910} C_DIS
LIN {X 0.001,Y -664.346,Z 962.509,A 0.000,B 0.000,C 90.000,E1 307.684} C_DIS
LIN {X -0.062,Y -664.637,Z 962.507,A 0.000,B 0.000,C 90.000,E1 307.202} C_DIS
LIN {X 0.131,Y -665.112,Z 962.499,A 0.000,B 0.000,C 90.000,E1 305.724} C_DIS
LIN {X -0.160,Y -665.367,Z 962.492,A 0.000,B 0.000,C 90.000,E1 304.532} C_DIS
LIN {X 0.303,Y -666.044,Z 962.481,A 0.000,B 0.000,C 90.000,E1 302.546} C_DIS
LIN {X 0.302,Y -667.677,Z 962.466,A 0.000,B 0.000,C 90.000,E1 299.873} C_DIS
LIN {X 0.010,Y -673.605,Z 962.442,A 0.000,B 0.000,C 90.000,E1 295.540} C_DIS
LIN {X 0.194,Y -676.244,Z 962.434,A 0.000,B 0.000,C 90.000,E1 294.079} C_DIS
LIN {X 0.038,Y -677.742,Z 962.429,A 0.000,B 0.000,C 90.000,E1 293.131} C_DIS
LIN {X 0.145,Y -678.284,Z 962.426,A 0.000,B 0.000,C 90.000,E1 292.642} C_DIS
LIN {X 0.260,Y -678.430,Z 962.423,A 0.000,B 0.000,C 90.000,E1 292.153} C_DIS
LIN {X -0.185,Y -678.223,Z 962.422,A 0.000,B 0.000,C 90.000,E1 291.950} C_DIS
LIN {X -0.070,Y -677.500,Z 962.419,A 0.000,B 0.000,C 90.000,E1 291.461} C_DIS
LIN {X -0.136,Y -676.435,Z 962.418,A 0.000,B 0.000,C 90.000,E1 291.227} C_DIS
LIN {X 0.042,Y -675.002,Z 962.417,A 0.000,B 0.000,C 90.000,E1 290.972} C_DIS
LIN {X -0.028,Y -673.146,Z 962.415,A 0.000,B 0.000,C 90.000,E1 290.737} C_DIS
LIN {X 0.054,Y -672.009,Z 962.415,A 0.000,B 0.000,C 90.000,E1 290.610} C_DIS
LIN {X 0.180,Y -668.846,Z 962.413,A 0.000,B 0.000,C 90.000,E1 290.375} C_DIS
LIN {X 0.092,Y -665.041,Z 962.412,A 0.000,B 0.000,C 90.000,E1 290.120} C_DIS
LIN {X -0.179,Y -658.941,Z 962.410,A 0.000,B 0.000,C 90.000,E1 289.758} C_DIS
LIN {X 0.006,Y -656.752,Z 962.409,A 0.000,B 0.000,C 90.000,E1 289.577} C_DIS
LIN {X -0.046,Y -656.725,Z 962.409,A 0.000,B 0.000,C 90.000,E1 289.577} C_DIS
LIN {X 0.057,Y -656.427,Z 962.408,A 0.000,B 0.000,C 90.000,E1 289.450} C_DIS
LIN {X 0.339,Y -656.889,Z 962.407,A 0.000,B 0.000,C 90.000,E1 289.141} C_DIS
LIN {X 0.170,Y -657.221,Z 962.406,A 0.000,B 0.000,C 90.000,E1 289.033} C_DIS
LIN {X 0.149,Y -659.550,Z 962.403,A 0.000,B 0.000,C 90.000,E1 288.544} C_DIS
LIN {X 0.090,Y -664.566,Z 962.398,A 0.000,B 0.000,C 90.000,E1 287.692} C_DIS
LIN {X -0.033,Y -667.919,Z 962.395,A 0.000,B 0.000,C 90.000,E1 287.094} C_DIS
LIN {X -0.131,Y -670.838,Z 962.392,A 0.000,B 0.000,C 90.000,E1 286.496} C_DIS
LIN {X -0.272,Y -672.888,Z 962.389,A 0.000,B 0.000,C 90.000,E1 286.024} C_DIS
LIN {X -0.214,Y -674.458,Z 962.386,A 0.000,B 0.000,C 90.000,E1 285.536} C_DIS
LIN {X 0.323,Y -675.821,Z 962.384,A 0.000,B 0.000,C 90.000,E1 285.009} C_DIS
LIN {X 0.221,Y -676.994,Z 962.381,A 0.000,B 0.000,C 90.000,E1 284.537} C_DIS
LIN {X 0.127,Y -677.983,Z 962.378,A 0.000,B 0.000,C 90.000,E1 284.064} C_DIS
LIN {X -0.043,Y -679.463,Z 962.373,A 0.000,B 0.000,C 90.000,E1 283.119} C_DIS
LIN {X -0.164,Y -680.227,Z 962.369,A 0.000,B 0.000,C 90.000,E1 282.411} C_DIS
LIN {X -0.383,Y -680.577,Z 962.366,A 0.000,B 0.000,C 90.000,E1 281.951} C_DIS
LIN {X 0.173,Y -680.652,Z 962.362,A 0.000,B 0.000,C 90.000,E1 281.186} C_DIS
LIN {X 0.095,Y -680.425,Z 962.360,A 0.000,B 0.000,C 90.000,E1 280.715} C_DIS
LIN {X -0.112,Y -679.992,Z 962.357,A 0.000,B 0.000,C 90.000,E1 280.254} C_DIS
LIN {X 0.310,Y -678.725,Z 962.353,A 0.000,B 0.000,C 90.000,E1 279.500} C_DIS
LIN {X 0.210,Y -677.558,Z 962.350,A 0.000,B 0.000,C 90.000,E1 279.029} C_DIS
LIN {X -0.005,Y -676.019,Z 962.348,A 0.000,B 0.000,C 90.000,E1 278.568} C_DIS
LIN {X -0.227,Y -674.239,Z 962.345,A 0.000,B 0.000,C 90.000,E1 278.106} C_DIS
LIN {X 0.210,Y -672.196,Z 962.342,A 0.000,B 0.000,C 90.000,E1 277.587} C_DIS
LIN {X -0.031,Y -669.784,Z 962.340,A 0.000,B 0.000,C 90.000,E1 277.125} C_DIS
LIN {X 0.362,Y -666.432,Z 962.336,A 0.000,B 0.000,C 90.000,E1 276.486} C_DIS
LIN {X 0.097,Y -664.075,Z 962.334,A 0.000,B 0.000,C 90.000,E1 276.144} C_DIS
LIN {X -0.106,Y -661.568,Z 962.332,A 0.000,B 0.000,C 90.000,E1 275.796} C_DIS
LIN {X 0.237,Y -657.909,Z 962.329,A 0.000,B 0.000,C 90.000,E1 275.277} C_DIS
LIN {X -0.156,Y -653.790,Z 962.327,A 0.000,B 0.000,C 90.000,E1 274.821} C_DIS
LIN {X 0.028,Y -648.092,Z 962.323,A 0.000,B 0.000,C 90.000,E1 274.188} C_DIS
LIN {X 0.304,Y -643.262,Z 962.321,A 0.000,B 0.000,C 90.000,E1 273.669} C_DIS
LIN {X 0.008,Y -638.195,Z 962.318,A 0.000,B 0.000,C 90.000,E1 273.212} C_DIS
LIN {X -0.053,Y -631.425,Z 962.315,A 0.000,B 0.000,C 90.000,E1 272.636} C_DIS
LIN {X 0.243,Y -624.382,Z 962.312,A 0.000,B 0.000,C 90.000,E1 272.064} C_DIS
LIN {X 0.201,Y -616.730,Z 962.309,A 0.000,B 0.000,C 90.000,E1 271.547} C_DIS
LIN {X -0.291,Y -610.512,Z 962.307,A 0.000,B 0.000,C 90.000,E1 271.203} C_DIS
LIN {X 0.191,Y -604.008,Z 962.305,A 0.000,B 0.000,C 90.000,E1 270.802} C_DIS
LIN {X -0.196,Y -597.269,Z 962.303,A 0.000,B 0.000,C 90.000,E1 270.516} C_DIS
LIN {X -0.212,Y -590.607,Z 962.301,A 0.000,B 0.000,C 90.000,E1 270.229} C_DIS
LIN {X 0.036,Y -583.287,Z 962.300,A 0.000,B 0.000,C 90.000,E1 269.943} C_DIS
LIN {X 0.019,Y -577.760,Z 962.299,A 0.000,B 0.000,C 90.000,E1 269.771} C_DIS
LIN {X 0.147,Y -571.940,Z 962.298,A 0.000,B 0.000,C 90.000,E1 269.599} C_DIS
LIN {X 0.050,Y -565.557,Z 962.297,A 0.000,B 0.000,C 90.000,E1 269.484} C_DIS
LIN {X 0.141,Y -558.034,Z 962.297,A 0.000,B 0.000,C 90.000,E1 269.370} C_DIS
LIN {X -0.236,Y -548.597,Z 962.296,A 0.000,B 0.000,C 90.000,E1 269.370} C_DIS
LIN {X -0.016,Y -546.261,Z 962.296,A 0.000,B 0.000,C 90.000,E1 269.312} C_DIS
LIN {X -0.035,Y -543.976,Z 962.296,A 0.000,B 0.000,C 90.000,E1 269.255} C_DIS
LIN {X -0.065,Y -543.820,Z 962.296,A 0.000,B 0.000,C 90.000,E1 269.255} C_DIS
LIN {X 0.009,Y -543.107,Z 962.295,A 0.000,B 0.000,C 90.000,E1 269.026} C_DIS
LIN {X 0.042,Y -540.652,Z 962.278,A 0.000,B 0.000,C 90.000,E1 266.045} C_DIS
LIN {X 0.242,Y -539.461,Z 962.269,A 0.000,B 0.000,C 90.000,E1 264.318} C_DIS
LIN {X -0.109,Y -538.371,Z 962.261,A 0.000,B 0.000,C 90.000,E1 262.932} C_DIS
LIN {X -0.008,Y -537.449,Z 962.254,A 0.000,B 0.000,C 90.000,E1 261.781} C_DIS
LIN {X 0.148,Y -536.296,Z 962.248,A 0.000,B 0.000,C 90.000,E1 260.622} C_DIS
LIN {X -0.150,Y -535.033,Z 962.242,A 0.000,B 0.000,C 90.000,E1 259.511} C_DIS
LIN {X 0.170,Y -532.925,Z 962.232,A 0.000,B 0.000,C 90.000,E1 257.757} C_DIS
LIN {X -0.211,Y -531.863,Z 962.227,A 0.000,B 0.000,C 90.000,E1 256.937} C_DIS
LIN {X 0.311,Y -529.484,Z 962.216,A 0.000,B 0.000,C 90.000,E1 254.866} C_DIS
LIN {X 0.066,Y -527.933,Z 962.208,A 0.000,B 0.000,C 90.000,E1 253.449} C_DIS
LIN {X 0.092,Y -526.287,Z 962.200,A 0.000,B 0.000,C 90.000,E1 252.000} C_DIS
LIN {X 0.255,Y -524.071,Z 962.190,A 0.000,B 0.000,C 90.000,E1 250.242} C_DIS
LIN {X 0.232,Y -522.598,Z 962.184,A 0.000,B 0.000,C 90.000,E1 249.082} C_DIS
LIN {X 0.004,Y -520.353,Z 962.174,A 0.000,B 0.000,C 90.000,E1 247.358} C_DIS
LIN {X -0.220,Y -518.167,Z 962.166,A 0.000,B 0.000,C 90.000,E1 245.921} C_DIS
LIN {X 0.072,Y -516.413,Z 962.160,A 0.000,B 0.000,C 90.000,E1 244.717} C_DIS
LIN {X 0.108,Y -513.644,Z 962.150,A 0.000,B 0.000,C 90.000,E1 242.948} C_DIS
LIN {X -0.249,Y -511.291,Z 962.142,A 0.000,B 0.000,C 90.000,E1 241.513} C_DIS
LIN {X -0.284,Y -509.324,Z 962.135,A 0.000,B 0.000,C 90.000,E1 240.333} C_DIS
LIN {X -0.093,Y -507.107,Z 962.128,A 0.000,B 0.000,C 90.000,E1 239.125} C_DIS
LIN {X 0.069,Y -504.732,Z 962.122,A 0.000,B 0.000,C 90.000,E1 237.916} C_DIS
LIN {X 0.189,Y -502.202,Z 962.115,A 0.000,B 0.000,C 90.000,E1 236.707} C_DIS
